MODE_NOTDEFINED:		
		resetAndDisable(alg:=algoritms.Auto_Avom_);
		resetAndDisable(alg:=algoritms.autoNu_1);
		resetAndDisable(alg:=algoritms.autoNu_2);
		resetAndDisable(alg:=algoritms.autoPns);
		resetAndDisable(alg:=algoritms.AUto_Ten_);
		resetAndDisable(alg:=algoritms.PNS_ON_MV_);
		resetAndDisable(alg:=algoritms.no);
		resetAndDisable(alg:=algoritms.ao);
		resetAndDisable(alg:=algoritms.Opres);
		resetAndDisable(alg:=algoritms.Pms);
		resetAndDisable(alg:=algoritms.dPmg);
		resetAndDisable(alg:=algoritms.ppu);
		resetAndDisable(alg:=algoritms.F1_1);
		resetAndDisable(alg:=algoritms.F1_2);
		resetAndDisable(alg:=algoritms.F2_Ch);
		resetAndDisable(alg:=algoritms.F2_R);
		resetAndDisable(alg:=algoritms.F3);
		resetAndDisable(alg:=algoritms.F4);
		resetAndDisable(alg:=algoritms.Kr6_Move);
		resetAndDisable(alg:=algoritms.AutoPNS_Start);
		resetAndDisable(alg:=algoritms.R_AutoAVom);
		resetAndDisable(alg:=algoritms.R_AutoTEN);
		resetAndDisable(alg:=algoritms.R_TestIM);
		resetAndDisable(alg:=algoritms.S_AutoAVOM);
		resetAndDisable(alg:=algoritms.S_AutoTEN);
		resetAndDisable(alg:=algoritms.S_Test_IM);
		resetAndDisable(alg:=algoritms.S_Vibr);
		resetAndDisable(alg:=algoritms.S_dPmg);
		resetAndDisable(alg:=algoritms.S_I);
		resetAndDisable(alg:=algoritms.S_K);
		resetAndDisable(alg:=algoritms.S_Pms);
		resetAndDisable(alg:=algoritms.S_V);
		resetAndDisable(alg:=algoritms.S_AP);
		resetAndDisable(alg:=algoritms.S_PP);
		resetAndDisable(alg:=algoritms.S_NO);
		resetAndDisable(alg:=algoritms.S_AO);
		resetAndDisable(alg:=algoritms.Test_IM);
		resetAndDisable(alg:=algoritms.Start_Test_P);
	resetAndDisable(alg:=algoritms.Test_P);
MODE_TESTIM:
		resetAndDisable(alg:=algoritms.Auto_Avom_);
		resetAndDisable(alg:=algoritms.autoNu_1);
		resetAndDisable(alg:=algoritms.autoNu_2);
		resetAndDisable(alg:=algoritms.autoPns);
		resetAndDisable(alg:=algoritms.AUto_Ten_);
		resetAndDisable(alg:=algoritms.PNS_ON_MV_);
		resetAndDisable(alg:=algoritms.Opres);
		resetAndDisable(alg:=algoritms.Pms);
		resetAndDisable(alg:=algoritms.dPmg);
		resetAndDisable(alg:=algoritms.no);
		resetAndDisable(alg:=algoritms.ao);
		resetAndDisable(alg:=algoritms.ppu);
		resetAndDisable(alg:=algoritms.F1_1);
		resetAndDisable(alg:=algoritms.F1_2);
		resetAndDisable(alg:=algoritms.F2_Ch);
		resetAndDisable(alg:=algoritms.F2_R);
		resetAndDisable(alg:=algoritms.F3);
		resetAndDisable(alg:=algoritms.F4);
		resetAndDisable(alg:=algoritms.Kr6_Move);
		resetAndDisable(alg:=algoritms.AutoPNS_Start);
		resetAndDisable(alg:=algoritms.R_AutoAVom);
		resetAndDisable(alg:=algoritms.R_AutoTEN);
		algoritms.R_TestIM.CanRun:=TRUE;
		resetAndDisable(alg:=algoritms.S_AutoAVOM);
		resetAndDisable(alg:=algoritms.S_AutoTEN);
		resetAndDisable(alg:=algoritms.S_Test_IM);
		resetAndDisable(alg:=algoritms.S_Vibr);
		resetAndDisable(alg:=algoritms.S_dPmg);
		resetAndDisable(alg:=algoritms.S_I);
		resetAndDisable(alg:=algoritms.S_K);
		resetAndDisable(alg:=algoritms.S_Pms);
		resetAndDisable(alg:=algoritms.S_V);
		resetAndDisable(alg:=algoritms.S_AP);
		resetAndDisable(alg:=algoritms.S_PP);
		algoritms.S_NO.CanRun:=TRUE;
		algoritms.S_AO.CanRun:=TRUE;
		resetAndDisable(alg:=algoritms.Start_Test_P);
		resetAndDisable(alg:=algoritms.Test_P);
MODE_PUSKV_R:
	resetAndDisable(alg:=algoritms.Auto_Avom_);
	resetAndDisable(alg:=algoritms.autoNu_1);
	resetAndDisable(alg:=algoritms.autoNu_2);
	resetAndDisable(alg:=algoritms.autoPns);
	resetAndDisable(alg:=algoritms.AUto_Ten_);
	resetAndDisable(alg:=algoritms.PNS_ON_MV_);
	resetAndDisable(alg:=algoritms.no);
		resetAndDisable(alg:=algoritms.ao);
	resetAndDisable(alg:=algoritms.Opres);
	resetAndDisable(alg:=algoritms.Pms);
	resetAndDisable(alg:=algoritms.dPmg);
	algoritms.ppu.CanRun:=TRUE;
	algoritms.ppu.run();
	resetAndDisable(alg:=algoritms.F1_2);
	resetAndDisable(alg:=algoritms.F2_Ch);
	resetAndDisable(alg:=algoritms.F2_R);
	resetAndDisable(alg:=algoritms.F3);
	resetAndDisable(alg:=algoritms.F4);
	resetAndDisable(alg:=algoritms.Kr6_Move);
	resetAndDisable(alg:=algoritms.AutoPNS_Start);
	resetAndDisable(alg:=algoritms.R_AutoAVom);
	resetAndDisable(alg:=algoritms.R_AutoTEN);
	resetAndDisable(alg:=algoritms.R_TestIM);
	resetAndDisable(alg:=algoritms.S_AutoAVOM);
	resetAndDisable(alg:=algoritms.S_AutoTEN);
	resetAndDisable(alg:=algoritms.S_Test_IM);
	resetAndDisable(alg:=algoritms.S_Vibr);
	resetAndDisable(alg:=algoritms.S_dPmg);
	resetAndDisable(alg:=algoritms.S_I);
	resetAndDisable(alg:=algoritms.S_K);
	resetAndDisable(alg:=algoritms.S_Pms);
	algoritms.S_V.CanRun:=FALSE;
	resetAndDisable(alg:=algoritms.S_PP);
	resetAndDisable(alg:=algoritms.S_AP);
	algoritms.S_NO.CanRun:=TRUE;
	algoritms.S_AO.CanRun:=TRUE;
	resetAndDisable(alg:=algoritms.Test_IM);
	reg_V:=TRUE;
	resetAndDisable(alg:=algoritms.Start_Test_P);
		resetAndDisable(alg:=algoritms.Test_P);
MODE_PUSKV_Ch:
	resetAndDisable(alg:=algoritms.Auto_Avom_);
	resetAndDisable(alg:=algoritms.autoNu_1);
	resetAndDisable(alg:=algoritms.autoNu_2);
	resetAndDisable(alg:=algoritms.autoPns);
	resetAndDisable(alg:=algoritms.AUto_Ten_);
	resetAndDisable(alg:=algoritms.PNS_ON_MV_);
	resetAndDisable(alg:=algoritms.no);
		resetAndDisable(alg:=algoritms.ao);
	resetAndDisable(alg:=algoritms.Opres);
	resetAndDisable(alg:=algoritms.Pms);
	resetAndDisable(alg:=algoritms.dPmg);
	algoritms.ppu.CanRun:=TRUE;
	algoritms.ppu.run();
	resetAndDisable(alg:=algoritms.F1_2);
	resetAndDisable(alg:=algoritms.F2_Ch);
	resetAndDisable(alg:=algoritms.F2_R);
	resetAndDisable(alg:=algoritms.F3);
	resetAndDisable(alg:=algoritms.F4);
	resetAndDisable(alg:=algoritms.Kr6_Move);
	resetAndDisable(alg:=algoritms.AutoPNS_Start);
	resetAndDisable(alg:=algoritms.R_AutoAVom);
	resetAndDisable(alg:=algoritms.R_AutoTEN);
	resetAndDisable(alg:=algoritms.R_TestIM);
	resetAndDisable(alg:=algoritms.S_AutoAVOM);
	resetAndDisable(alg:=algoritms.S_AutoTEN);
	resetAndDisable(alg:=algoritms.S_Test_IM);
	resetAndDisable(alg:=algoritms.S_Vibr);
	resetAndDisable(alg:=algoritms.S_dPmg);
	resetAndDisable(alg:=algoritms.S_I);
	resetAndDisable(alg:=algoritms.S_K);
	resetAndDisable(alg:=algoritms.S_Pms);
	algoritms.S_V.CanRun:=FALSE;
	resetAndDisable(alg:=algoritms.S_PP);
	resetAndDisable(alg:=algoritms.S_AP);
	algoritms.S_NO.CanRun:=TRUE;
	algoritms.S_AO.CanRun:=TRUE;
	resetAndDisable(alg:=algoritms.Test_IM);
	reg_V:=TRUE;
	resetAndDisable(alg:=algoritms.Start_Test_P);
		resetAndDisable(alg:=algoritms.Test_P);
MODE_PUSKK:
	resetAndDisable(alg:=algoritms.Auto_Avom_);
	resetAndDisable(alg:=algoritms.autoNu_1);
	resetAndDisable(alg:=algoritms.autoNu_2);
	resetAndDisable(alg:=algoritms.autoPns);
	resetAndDisable(alg:=algoritms.AUto_Ten_);
	resetAndDisable(alg:=algoritms.PNS_ON_MV_);
	resetAndDisable(alg:=algoritms.no);
		resetAndDisable(alg:=algoritms.ao);
	resetAndDisable(alg:=algoritms.Opres);
	resetAndDisable(alg:=algoritms.Pms);
	resetAndDisable(alg:=algoritms.dPmg);
	algoritms.ppu.CanRun:=TRUE;
	algoritms.ppu.run();
	resetAndDisable(alg:=algoritms.F1_2);
	resetAndDisable(alg:=algoritms.F2_Ch);
	resetAndDisable(alg:=algoritms.F2_R);
	resetAndDisable(alg:=algoritms.F3);
	resetAndDisable(alg:=algoritms.F4);
	resetAndDisable(alg:=algoritms.Kr6_Move);
	resetAndDisable(alg:=algoritms.AutoPNS_Start);
	resetAndDisable(alg:=algoritms.R_AutoAVom);
	resetAndDisable(alg:=algoritms.R_AutoTEN);
	resetAndDisable(alg:=algoritms.R_TestIM);
	resetAndDisable(alg:=algoritms.S_AutoAVOM);
	resetAndDisable(alg:=algoritms.S_AutoTEN);
	resetAndDisable(alg:=algoritms.S_Test_IM);
	resetAndDisable(alg:=algoritms.S_Vibr);
	resetAndDisable(alg:=algoritms.S_dPmg);
	resetAndDisable(alg:=algoritms.S_I);
	algoritms.S_K.CanRun:=FALSE;
	resetAndDisable(alg:=algoritms.S_Pms);
	resetAndDisable(alg:=algoritms.S_V);
	resetAndDisable(alg:=algoritms.S_PP);
	resetAndDisable(alg:=algoritms.S_AP);
	algoritms.S_NO.CanRun:=TRUE;
	algoritms.S_AO.CanRun:=TRUE;
	resetAndDisable(alg:=algoritms.Test_IM);
	resetAndDisable(alg:=algoritms.Start_Test_P);
		resetAndDisable(alg:=algoritms.Test_P);
MODE_PROVPMS:
	resetAndDisable(alg:=algoritms.Auto_Avom_);
	resetAndDisable(alg:=algoritms.autoNu_1);
	resetAndDisable(alg:=algoritms.autoNu_2);
	resetAndDisable(alg:=algoritms.autoPns);
	resetAndDisable(alg:=algoritms.AUto_Ten_);
	resetAndDisable(alg:=algoritms.PNS_ON_MV_);
	resetAndDisable(alg:=algoritms.no);
		resetAndDisable(alg:=algoritms.ao);
	resetAndDisable(alg:=algoritms.Opres);
	resetAndDisable(alg:=algoritms.Pms);
	resetAndDisable(alg:=algoritms.dPmg);
	resetAndDisable(alg:=algoritms.ppu);
	resetAndDisable(alg:=algoritms.F1_2);
	resetAndDisable(alg:=algoritms.F2_Ch);
	resetAndDisable(alg:=algoritms.F2_R);
	resetAndDisable(alg:=algoritms.F3);
	resetAndDisable(alg:=algoritms.F4);
	resetAndDisable(alg:=algoritms.Kr6_Move);
	resetAndDisable(alg:=algoritms.AutoPNS_Start);
	resetAndDisable(alg:=algoritms.R_AutoAVom);
	resetAndDisable(alg:=algoritms.R_AutoTEN);
	resetAndDisable(alg:=algoritms.R_TestIM);
	resetAndDisable(alg:=algoritms.S_AutoAVOM);
	resetAndDisable(alg:=algoritms.S_AutoTEN);
	resetAndDisable(alg:=algoritms.S_Test_IM);
	resetAndDisable(alg:=algoritms.S_Vibr);
	resetAndDisable(alg:=algoritms.S_dPmg);
	resetAndDisable(alg:=algoritms.S_I);
	resetAndDisable(alg:=algoritms.S_K);
	algoritms.S_Pms.CanRun:=FALSE;
	resetAndDisable(alg:=algoritms.S_V);
	resetAndDisable(alg:=algoritms.S_PP);
	resetAndDisable(alg:=algoritms.S_AP);
	algoritms.S_NO.CanRun:=TRUE;
	algoritms.S_AO.CanRun:=TRUE;
	resetAndDisable(alg:=algoritms.Test_IM);
	resetAndDisable(alg:=algoritms.Start_Test_P);
		resetAndDisable(alg:=algoritms.Test_P);
MODE_PROBDPMG:
	resetAndDisable(alg:=algoritms.Auto_Avom_);
	resetAndDisable(alg:=algoritms.autoNu_1);
	resetAndDisable(alg:=algoritms.autoNu_2);
	resetAndDisable(alg:=algoritms.autoPns);
	resetAndDisable(alg:=algoritms.AUto_Ten_);
	resetAndDisable(alg:=algoritms.PNS_ON_MV_);
	resetAndDisable(alg:=algoritms.no);
		resetAndDisable(alg:=algoritms.ao);
	resetAndDisable(alg:=algoritms.Opres);
	resetAndDisable(alg:=algoritms.Pms);
	resetAndDisable(alg:=algoritms.dPmg);
	resetAndDisable(alg:=algoritms.ppu);
	resetAndDisable(alg:=algoritms.F1_2);
	resetAndDisable(alg:=algoritms.F2_Ch);
	resetAndDisable(alg:=algoritms.F2_R);
	resetAndDisable(alg:=algoritms.F3);
	resetAndDisable(alg:=algoritms.F4);
	resetAndDisable(alg:=algoritms.Kr6_Move);
	resetAndDisable(alg:=algoritms.AutoPNS_Start);
	resetAndDisable(alg:=algoritms.R_AutoAVom);
	resetAndDisable(alg:=algoritms.R_AutoTEN);
	resetAndDisable(alg:=algoritms.R_TestIM);
	resetAndDisable(alg:=algoritms.S_AutoAVOM);
	resetAndDisable(alg:=algoritms.S_AutoTEN);
	resetAndDisable(alg:=algoritms.S_Test_IM);
	resetAndDisable(alg:=algoritms.S_Vibr);
	resetAndDisable(alg:=algoritms.S_Pms);
	resetAndDisable(alg:=algoritms.S_I);
	resetAndDisable(alg:=algoritms.S_K);
	algoritms.S_dPmg.CanRun:=FALSE;
	resetAndDisable(alg:=algoritms.S_V);
	resetAndDisable(alg:=algoritms.S_PP);
	resetAndDisable(alg:=algoritms.S_AP);
	algoritms.S_NO.CanRun:=TRUE;
	algoritms.S_AO.CanRun:=TRUE;
	resetAndDisable(alg:=algoritms.Test_IM);
resetAndDisable(alg:=algoritms.Start_Test_P);
		resetAndDisable(alg:=algoritms.Test_P);
MODE_I:
	resetAndDisable(alg:=algoritms.Auto_Avom_);
	resetAndDisable(alg:=algoritms.autoNu_1);
	resetAndDisable(alg:=algoritms.autoNu_2);
	resetAndDisable(alg:=algoritms.autoPns);
	resetAndDisable(alg:=algoritms.AUto_Ten_);
	resetAndDisable(alg:=algoritms.PNS_ON_MV_);
	resetAndDisable(alg:=algoritms.no);
		resetAndDisable(alg:=algoritms.ao);
	resetAndDisable(alg:=algoritms.Opres);
	resetAndDisable(alg:=algoritms.Pms);
	resetAndDisable(alg:=algoritms.dPmg);
	algoritms.ppu.CanRun:=TRUE;
	algoritms.ppu.run();
	resetAndDisable(alg:=algoritms.F1_2);
	resetAndDisable(alg:=algoritms.F2_Ch);
	resetAndDisable(alg:=algoritms.F2_R);
	resetAndDisable(alg:=algoritms.F3);
	resetAndDisable(alg:=algoritms.F4);
	resetAndDisable(alg:=algoritms.Kr6_Move);
	resetAndDisable(alg:=algoritms.AutoPNS_Start);
	resetAndDisable(alg:=algoritms.R_AutoAVom);
	resetAndDisable(alg:=algoritms.R_AutoTEN);
	resetAndDisable(alg:=algoritms.R_TestIM);
	resetAndDisable(alg:=algoritms.S_AutoAVOM);
	resetAndDisable(alg:=algoritms.S_AutoTEN);
	resetAndDisable(alg:=algoritms.S_Test_IM);
	resetAndDisable(alg:=algoritms.S_Vibr);
	resetAndDisable(alg:=algoritms.S_Pms);
	resetAndDisable(alg:=algoritms.S_dPmg);
	resetAndDisable(alg:=algoritms.S_K);
	algoritms.S_I.CanRun:=FALSE;
	resetAndDisable(alg:=algoritms.S_V);
	resetAndDisable(alg:=algoritms.S_PP);
	resetAndDisable(alg:=algoritms.S_AP);
	algoritms.S_NO.CanRun:=TRUE;
	algoritms.S_AO.CanRun:=TRUE;
	resetAndDisable(alg:=algoritms.Test_IM);
	resetAndDisable(alg:=algoritms.Start_Test_P);
		resetAndDisable(alg:=algoritms.Test_P);
MODE_O:
	resetAndDisable(alg:=algoritms.Auto_Avom_);
	resetAndDisable(alg:=algoritms.autoNu_1);
	resetAndDisable(alg:=algoritms.autoNu_2);
	resetAndDisable(alg:=algoritms.autoPns);
	resetAndDisable(alg:=algoritms.AUto_Ten_);
	resetAndDisable(alg:=algoritms.PNS_ON_MV_);
	resetAndDisable(alg:=algoritms.no);
		resetAndDisable(alg:=algoritms.ao);
	resetAndDisable(alg:=algoritms.S_I);
	resetAndDisable(alg:=algoritms.Pms);
	resetAndDisable(alg:=algoritms.dPmg);
	resetAndDisable(alg:=algoritms.ppu);
	resetAndDisable(alg:=algoritms.F1_1);
	resetAndDisable(alg:=algoritms.F1_2);
	resetAndDisable(alg:=algoritms.F2_Ch);
	resetAndDisable(alg:=algoritms.F2_R);
	resetAndDisable(alg:=algoritms.F3);
	resetAndDisable(alg:=algoritms.F4);
	resetAndDisable(alg:=algoritms.Kr6_Move);
	resetAndDisable(alg:=algoritms.AutoPNS_Start);
	resetAndDisable(alg:=algoritms.R_AutoAVom);
	resetAndDisable(alg:=algoritms.R_AutoTEN);
	resetAndDisable(alg:=algoritms.R_TestIM);
	resetAndDisable(alg:=algoritms.S_AutoAVOM);
	resetAndDisable(alg:=algoritms.S_AutoTEN);
	resetAndDisable(alg:=algoritms.S_Test_IM);
	resetAndDisable(alg:=algoritms.S_Vibr);
	resetAndDisable(alg:=algoritms.S_Pms);
	resetAndDisable(alg:=algoritms.S_dPmg);
	resetAndDisable(alg:=algoritms.S_K);
	algoritms.Opres.CanRun:=FALSE;
	resetAndDisable(alg:=algoritms.S_V);
	resetAndDisable(alg:=algoritms.S_PP);
	resetAndDisable(alg:=algoritms.S_AP);
	algoritms.S_NO.CanRun:=TRUE;
	algoritms.S_AO.CanRun:=TRUE;
	resetAndDisable(alg:=algoritms.Test_IM);
	resetAndDisable(alg:=algoritms.Start_Test_P);
		resetAndDisable(alg:=algoritms.Test_P);
		
TEST_PROTECTIONS:	
		resetAndDisable(alg:=algoritms.Auto_Avom_);
		resetAndDisable(alg:=algoritms.autoNu_1);
		resetAndDisable(alg:=algoritms.autoNu_2);
		resetAndDisable(alg:=algoritms.autoPns);
		resetAndDisable(alg:=algoritms.AUto_Ten_);
		resetAndDisable(alg:=algoritms.PNS_ON_MV_);
		algoritms.no.CanRun:=TRUE;
		algoritms.ao.CanRun:=TRUE;
		resetAndDisable(alg:=algoritms.Opres);
		resetAndDisable(alg:=algoritms.Pms);
		resetAndDisable(alg:=algoritms.dPmg);
		resetAndDisable(alg:=algoritms.ppu);
		resetAndDisable(alg:=algoritms.F1_1);
		resetAndDisable(alg:=algoritms.F1_2);
		resetAndDisable(alg:=algoritms.F2_Ch);
		resetAndDisable(alg:=algoritms.F2_R);
		resetAndDisable(alg:=algoritms.F3);
		resetAndDisable(alg:=algoritms.F4);
		resetAndDisable(alg:=algoritms.Kr6_Move);
		resetAndDisable(alg:=algoritms.AutoPNS_Start);
		resetAndDisable(alg:=algoritms.R_AutoAVom);
		resetAndDisable(alg:=algoritms.R_AutoTEN);
		resetAndDisable(alg:=algoritms.R_TestIM);
		resetAndDisable(alg:=algoritms.S_AutoAVOM);
		resetAndDisable(alg:=algoritms.S_AutoTEN);
		resetAndDisable(alg:=algoritms.S_Test_IM);
		resetAndDisable(alg:=algoritms.S_Vibr);
		resetAndDisable(alg:=algoritms.S_dPmg);
		resetAndDisable(alg:=algoritms.S_I);
		resetAndDisable(alg:=algoritms.S_K);
		resetAndDisable(alg:=algoritms.S_Pms);
		resetAndDisable(alg:=algoritms.S_V);
		resetAndDisable(alg:=algoritms.S_AP);
		resetAndDisable(alg:=algoritms.S_PP);
		algoritms.S_NO.CanRun:=TRUE;
		algoritms.S_AO.CanRun:=TRUE;
		resetAndDisable(alg:=algoritms.Test_IM);
		Reset_ALL_P ();
		resetAndDisable(alg:=algoritms.Start_Test_P);
		algoritms.Test_P.CanRun:=TRUE;
		algoritms.Test_P.EnableOpcControl();

END_CASE

END_IF
END_METHOD

METHOD PUBLIC resetAndDisable
VAR_INPUT
	alg:REFERENCE TO BaseAlgoritm;
END_VAR
IF __ISVALIDREF(alg) THEN
	IF alg.isRuning THEN
		alg.reset();
	END_IF
	alg.CanRun:=FALSE;
END_IF
END_METHOD

END_FUNCTION_BLOCK

// lowLevel_ecl/algoritms/BaseAlgoritmsManager
	{attribute 'symbol' := 'none'}
FUNCTION_BLOCK BaseAlgoritmsManager EXTENDS BaseAlgoritm
VAR_INPUT
END_VAR
VAR_OUTPUT
END_VAR
VAR

END_VAR

SUPER^();
callBase();

METHOD PROTECTED onInit
VAR_INPUT
END_VAR
SUPER^.onInit();
onStart();
END_METHOD

METHOD PROTECTED onStart
VAR_INPUT
END_VAR
END_METHOD

METHOD PROTECTED processCmd;
VAR_INPUT
	cmd:UINT;
	sender:UINT;
	parametr:UINT;
END_VAR
END_METHOD

END_FUNCTION_BLOCK

// K1/std12k5/Narabotka/NO
	{attribute 'symbol' := 'none'}
FUNCTION_BLOCK NO EXTENDS BaseIM
VAR_INPUT
END_VAR
VAR_OUTPUT
	
		{attribute 'symbol' := 'read'}
	narabotka:UDINT;
END_VAR
VAR
	flag:BOOL;
	Work_END:F_TRIG;
	
	AvomStartted:R_TRIG;
END_VAR

SUPER^();
Work_END (CLK:=(algmanager.mode=modegpa.MODE_WORK_K OR algmanager.mode=modegpa.MODE_WORK_M));
IF Work_END.Q THEN
	flag:=TRUE;
END_IF
AvomStartted(CLK:=(algmanager.mode=modegpa.MODE_NO) AND flag);
IF AvomStartted.Q THEN
	narabotka:= narabotka + 1;
	SaveToFile();
	flag:=FALSE;
END_IF

METHOD PROTECTED readPersistent
VAR_INPUT
END_VAR

narabotka:=STRING_TO_UDINT(readValue());
END_METHOD

METHOD PROTECTED writePersistent
VAR_INPUT
END_VAR

writeValue(value:= UDINT_TO_STRING(narabotka),'Наработка');
END_METHOD

END_FUNCTION_BLOCK

// K2/std12k5/Natabotka/NO
	{attribute 'symbol' := 'none'}
FUNCTION_BLOCK NO EXTENDS BaseIM
VAR_INPUT
END_VAR
VAR_OUTPUT
	
		{attribute 'symbol' := 'read'}
	narabotka:UDINT;
END_VAR
VAR
	flag:BOOL;
	Work_END:F_TRIG;
	
	AvomStartted:R_TRIG;
END_VAR

SUPER^();
Work_END (CLK:=(algmanager.mode=modegpa.MODE_WORK_K OR algmanager.mode=modegpa.MODE_WORK_M));
IF Work_END.Q THEN
	flag:=TRUE;
END_IF
AvomStartted(CLK:=(algmanager.mode=modegpa.MODE_NO) AND flag);
IF AvomStartted.Q THEN
	narabotka:= narabotka + 1;
	SaveToFile();
	flag:=FALSE;
END_IF

METHOD PROTECTED readPersistent
VAR_INPUT
END_VAR

narabotka:=STRING_TO_UDINT(readValue());
END_METHOD

METHOD PROTECTED writePersistent
VAR_INPUT
END_VAR

writeValue(value:= UDINT_TO_STRING(narabotka),'Наработка');
END_METHOD

END_FUNCTION_BLOCK

// K1/std12k5/Narabotka/AO
	{attribute 'symbol' := 'none'}
FUNCTION_BLOCK AO EXTENDS BaseIM
VAR_INPUT
END_VAR
VAR_OUTPUT
	
		{attribute 'symbol' := 'read'}
	narabotka:UDINT;
END_VAR
VAR
	Work_End:F_TRIG;
	flag:bool;
	
	AvomStartted:R_TRIG;
END_VAR

SUPER^();
Work_END (CLK:=(algmanager.mode=modegpa.MODE_WORK_K OR algmanager.mode=modegpa.MODE_WORK_M));
IF Work_END.Q THEN
	flag:=TRUE;
END_IF
AvomStartted(CLK:=(algmanager.mode=modegpa.MODE_AO) AND flag);
IF AvomStartted.Q THEN
	narabotka:= narabotka + 1;
	SaveToFile();
	flag:=false;
END_IF

METHOD PROTECTED readPersistent
VAR_INPUT
END_VAR

narabotka:=STRING_TO_UDINT(readValue());
END_METHOD

METHOD PROTECTED writePersistent
VAR_INPUT
END_VAR

writeValue(value:= UDINT_TO_STRING(narabotka),'Наработка');
END_METHOD

END_FUNCTION_BLOCK

// K2/std12k5/Natabotka/AO
	{attribute 'symbol' := 'none'}
FUNCTION_BLOCK AO EXTENDS BaseIM
VAR_INPUT
END_VAR
VAR_OUTPUT
	
		{attribute 'symbol' := 'read'}
	narabotka:UDINT;
END_VAR
VAR
	Work_End:F_TRIG;
	flag:bool;
	
	AvomStartted:R_TRIG;
END_VAR

SUPER^();
Work_END (CLK:=(algmanager.mode=modegpa.MODE_WORK_K OR algmanager.mode=modegpa.MODE_WORK_M));
IF Work_END.Q THEN
	flag:=TRUE;
END_IF
AvomStartted(CLK:=(algmanager.mode=modegpa.MODE_AO) AND flag);
IF AvomStartted.Q THEN
	narabotka:= narabotka + 1;
	SaveToFile();
	flag:=false;
END_IF

METHOD PROTECTED readPersistent
VAR_INPUT
END_VAR

narabotka:=STRING_TO_UDINT(readValue());
END_METHOD

METHOD PROTECTED writePersistent
VAR_INPUT
END_VAR

writeValue(value:= UDINT_TO_STRING(narabotka),'Наработка');
END_METHOD

END_FUNCTION_BLOCK

// K2/std12k5/Prov/Reset_ALL_P
FUNCTION Reset_ALL_P : BOOL
VAR_INPUT
END_VAR
VAR
END_VAR


		Protections.p_TOpornogoPodshipnikaEDT_1.reset ();
		Protections.p_TOpornoYpornogoPodshipnikaEDT_2.reset ();
		Protections.p_TOpornoYpornogoPodshipnikaKolesaRedEDT_3.reset ();
		Protections.p_TOpornoYpornogoPodshipnikaKolesaRedHT_4.reset ();
		Protections.p_TOpornogoPodshipnikaShesterniReduktoraT_5.reset ();
		Protections.p_TOpornogoPodshipnikaReduktoraHT_6.reset ();
		Protections.p_TOpornoYpornogoPodshipnikaNagnetateljaT_7.reset ();
		Protections.p_TOpornoYpornogoPodshipnikaSvobodnogoKoncaNT_8.reset ();
		Protections.p_TYpornogoPodshipnikaRavKolodokHT_9.reset ();
		Protections.p_TYpornogoPodshipnikaNerabKolodokHT_10.reset ();
		Protections.p_TgazaNaVyhodeH.reset ();
		
	(*Давления*)
		
		Protections.p_OsSdvigNagnetatelja_Plus.reset ();
		Protections.p_OsSdvigNagnetatelja_Minus.reset ();
		Protections.p_DGazaNaVhodeNagnetatelja_GPA_STOP.reset ();
		Protections.p_DGazaNaVyhodeNagnetatelja_GPA_STOP.reset ();
		//p_DGazaNaVhodeNagnetatelja:AiProtection (table:=protectManager.getTable())							:=(ai:=ai.DGazaNaVhodeNagnetatelja,controlLimit:=statusAi.LA,delay:=(value:=T#3S));
		Protections.p_DGazaNaVyhodeNagnetatelja.reset ();
		Protections.p_PerepadDavlenieMasloGaz.reset ();
		Protections.p_DavlenijaMasloSmNizkoe.reset ();
		Protections.p_DavlenijaMasloSmVysokoe.reset ();
	
	(*Вибрация*)
		
		Protections.p_VibroSkorostOPED_T1.reset ();
		Protections.p_VibroSkorostOYPED_T2.reset ();
		Protections.p_VibroSkorostOYPKolesaED_T3.reset ();
		Protections.p_VibroSkorostOPKolesaRH_T4.reset ();
		Protections.p_VibroSkorostOPShesterniRED_T5.reset ();
		Protections.p_VibroSkorostOPShesterniReduktoraH_T6.reset ();
	(*Дискретные сигналы *)
		
		Protections.p_PerepadDavlenieMasloGaz_Less100.reset ();
		Protections.p_RegVozbOff.reset ();
		Protections.p_Fail_Chastotniy_Pusk.reset ();
		Protections.p_OFFAvarSwitch.reset ();
		Protections.p_AOKC_SHKC.reset ();
		Protections.p_AO_PRU.reset ();
		Protections.p_AO_fromSHU.reset ();
					
(*Защиты по ИМ *)																							
		Protections.p_mvOff.reset ();
		Protections.p_kran1.reset ();
		Protections.p_kran2.reset ();

END_FUNCTION

// LowLevel_Algoritms/algoritms/AiProtection
	{attribute 'symbol' := 'none'}
FUNCTION_BLOCK AiProtection EXTENDS BaseProtection
VAR_INPUT
	ai:REFERENCE TO AISource;
	controlLimit:statusAi;
	ControlValue:REAL;
	{attribute 'symbol' := 'read'}
	delay:TimeParametr(table:=ADR(objectTable));	
END_VAR
VAR_OUTPUT
END_VAR
VAR
	flag:bool;
	timer:TON;
	timer2:ton;
END_VAR

SUPER^();
IF __ISVALIDREF(ai) THEN
	IF	((ai.interval = controlLimit) AND (ControlValue = 0)) OR ((ai.interval >= controlLimit) AND (ControlValue <> 0)) THEN
		flag:=TRUE;
	ELSE
		flag:=FALSE;
	END_IF
	IF	ControlValue <> 0 THEN
		timer2 (in:= (flag AND (ai.value >= ControlValue)), pt:=delay.Value);
		IF	timer2.Q THEN
			signaling:=TRUE;
		ELSE
			signaling:=FALSE;
		END_IF
	ELSE
		timer(IN:=flag,PT:=delay.Value);
		IF timer.Q THEN
			signaling:=TRUE;
		ELSE
			signaling:=FALSE;
		END_IF
	END_IF
END_IF

METHOD PUBLIC reset
VAR_INPUT
END_VAR
SUPER^.reset();
timer(in:=FALSE);
signaling:=FALSE;
DisableAiLimits( ai,getLimitFlags(controlLimit));
END_METHOD

METHOD PUBLIC run
VAR_INPUT
END_VAR
SUPER^.run();
EnableAiLimits( ai,getLimitFlags(controlLimit));
END_METHOD

END_FUNCTION_BLOCK

// LowLevel_Algoritms/Common/DisableAiLimits
FUNCTION DisableAiLimits : Bool
VAR_INPUT
	ai:REFERENCE TO AISource;
	flags:BYTE;
END_VAR
VAR
END_VAR

IF __ISVALIDREF(ai) THEN
	ai.disabledAlarms:=ai.disabledAlarms OR flags;
END_IF

END_FUNCTION

// LowLevel_Algoritms/Common/getLimitFlags
FUNCTION getLimitFlags : BYTE
VAR_INPUT
	AiLimit:statusAi;
END_VAR
VAR
END_VAR

CASE AiLimit OF
	statusAi.LW, statusAi.LA:
		getLimitFlags:=AnalogAlarms.LW OR AnalogAlarms.LA;
	statusAi.HW,statusAi.HA:
		getLimitFlags:=AnalogAlarms.HW OR AnalogAlarms.HA;
ELSE
	getLimitFlags:=0;
END_CASE

END_FUNCTION

// LowLevel_Algoritms/Common/EnableAiLimits
FUNCTION EnableAiLimits : Bool
VAR_INPUT
	ai:REFERENCE TO AISource;
	flags:BYTE;
END_VAR
VAR
END_VAR

IF __ISVALIDREF(ai) THEN
	ai.disabledAlarms:=ai.disabledAlarms AND (flags XOR 16#FF);
END_IF

END_FUNCTION

// K1/std12k5/Prov/Reset_ALL_P
FUNCTION Reset_ALL_P : BOOL
VAR_INPUT
END_VAR
VAR
END_VAR


		Protections.p_TOpornogoPodshipnikaEDT_1.reset ();
		Protections.p_TOpornoYpornogoPodshipnikaEDT_2.reset ();
		Protections.p_TOpornoYpornogoPodshipnikaKolesaRedEDT_3.reset ();
		Protections.p_TOpornoYpornogoPodshipnikaKolesaRedHT_4.reset ();
		Protections.p_TOpornogoPodshipnikaShesterniReduktoraT_5.reset ();
		Protections.p_TOpornogoPodshipnikaReduktoraHT_6.reset ();
		Protections.p_TOpornoYpornogoPodshipnikaNagnetateljaT_7.reset ();
		Protections.p_TOpornoYpornogoPodshipnikaSvobodnogoKoncaNT_8.reset ();
		Protections.p_TYpornogoPodshipnikaRavKolodokHT_9.reset ();
		Protections.p_TYpornogoPodshipnikaNerabKolodokHT_10.reset ();
		Protections.p_TgazaNaVyhodeH.reset ();
		
	(*Давления*)
		
		Protections.p_OsSdvigNagnetatelja_Plus.reset ();
		Protections.p_OsSdvigNagnetatelja_Minus.reset ();
		Protections.p_DGazaNaVhodeNagnetatelja_GPA_STOP.reset ();
		Protections.p_DGazaNaVyhodeNagnetatelja_GPA_STOP.reset ();
		//p_DGazaNaVhodeNagnetatelja:AiProtection (table:=protectManager.getTable())							:=(ai:=ai.DGazaNaVhodeNagnetatelja,controlLimit:=statusAi.LA,delay:=(value:=T#3S));
		Protections.p_DGazaNaVyhodeNagnetatelja.reset ();
		Protections.p_PerepadDavlenieMasloGaz.reset ();
		Protections.p_DavlenijaMasloSmNizkoe.reset ();
		Protections.p_DavlenijaMasloSmVysokoe.reset ();
	
	(*Вибрация*)
		
		Protections.p_VibroSkorostOPED_T1.reset ();
		Protections.p_VibroSkorostOYPED_T2.reset ();
		Protections.p_VibroSkorostOYPKolesaED_T3.reset ();
		Protections.p_VibroSkorostOPKolesaRH_T4.reset ();
		Protections.p_VibroSkorostOPShesterniRED_T5.reset ();
		Protections.p_VibroSkorostOPShesterniReduktoraH_T6.reset ();
	(*Дискретные сигналы *)
		
		Protections.p_PerepadDavlenieMasloGaz_Less100.reset ();
		Protections.p_RegVozbOff.reset ();
		Protections.p_Fail_Chastotniy_Pusk.reset ();
		Protections.p_OFFAvarSwitch.reset ();
		Protections.p_AOKC_SHKC.reset ();
		Protections.p_AO_PRU.reset ();
		Protections.p_AO_fromSHU.reset ();
					
(*Защиты по ИМ *)																							
		Protections.p_mvOff.reset ();
		Protections.p_kran1.reset ();
		Protections.p_kran2.reset ();

END_FUNCTION

// K1/std12k5/Prov/Test_Protections
	{attribute 'symbol' := 'none'}
FUNCTION_BLOCK  Test_Protections EXTENDS BaseAlgoritm
VAR_INPUT
	{attribute 'symbol' := 'read'}
	Protect_On_1:DiscretParametr(table:=ADR(objectTable));//{name:маска ввключения защит}
	{attribute 'symbol' := 'read'}
	Protect_On_2:DiscretParametr(table:=ADR(objectTable));//{name:маска ввключения защит}
	{attribute 'symbol' := 'read'}
	Protect_On_3:DiscretParametr(table:=ADR(objectTable));//{name:маска ввключения защит}
	{attribute 'symbol' := 'read'}
	Protect_On_4:DiscretParametr(table:=ADR(objectTable));//{name:маска ввключения защит}
	{attribute 'symbol' := 'read'}
	AO_start:DiscretParametr(table:=ADR(objectTable));//{name:маска ввключения защит}
END_VAR
VAR_OUTPUT
	
END_VAR
VAR

	
	
END_VAR

SUPER^();
Run_Protection(Protections.p_TOpornogoPodshipnikaEDT_1						, 1		,Protect_On_1.value);
Run_Protection(Protections.p_TOpornoYpornogoPodshipnikaEDT_2				, 2		,Protect_On_1.value);
Run_Protection(Protections.p_TOpornoYpornogoPodshipnikaKolesaRedEDT_3  		, 4		,Protect_On_1.value);
Run_Protection(Protections.p_TOpornoYpornogoPodshipnikaKolesaRedHT_4   		, 8		,Protect_On_1.value);
Run_Protection(Protections.p_TOpornogoPodshipnikaShesterniReduktoraT_5	 	, 16	,Protect_On_1.value);
Run_Protection(Protections.p_TOpornogoPodshipnikaReduktoraHT_6	         	, 32	,Protect_On_1.value);
Run_Protection(Protections.p_TOpornoYpornogoPodshipnikaNagnetateljaT_7	 	, 64	,Protect_On_1.value);
Run_Protection(Protections.p_TOpornoYpornogoPodshipnikaSvobodnogoKoncaNT_8	, 128	,Protect_On_1.value);
Run_Protection(Protections.p_TYpornogoPodshipnikaRavKolodokHT_9				, 256	,Protect_On_1.value);
Run_Protection(Protections.p_TYpornogoPodshipnikaNerabKolodokHT_10			, 512	,Protect_On_1.value);
Run_Protection(Protections.p_TgazaNaVyhodeH									, 1		,Protect_On_2.value);
Run_Protection(Protections.p_OsSdvigNagnetatelja_Plus						, 2		,Protect_On_2.value);
Run_Protection(Protections.p_OsSdvigNagnetatelja_Minus						, 4		,Protect_On_2.value);
Run_Protection(Protections.p_DGazaNaVhodeNagnetatelja_GPA_STOP				, 8		,Protect_On_2.value);
Run_Protection(Protections.p_DGazaNaVyhodeNagnetatelja_GPA_STOP				, 16	,Protect_On_2.value);
Run_Protection(Protections.p_DGazaNaVyhodeNagnetatelja						, 32	,Protect_On_2.value);
Run_Protection(Protections.p_PerepadDavlenieMasloGaz						, 64	,Protect_On_2.value);
Run_Protection(Protections.p_DavlenijaMasloSmNizkoe							, 128	,Protect_On_2.value);
Run_Protection(Protections.p_DavlenijaMasloSmVysokoe						, 256	,Protect_On_2.value);
Run_Protection(Protections.p_VibroSkorostOPED_T1							, 512	,Protect_On_2.value);
Run_Protection(Protections.p_VibroSkorostOYPED_T2							, 1		,Protect_On_3.value);
Run_Protection(Protections.p_VibroSkorostOYPKolesaED_T3						, 2		,Protect_On_3.value);
Run_Protection(Protections.p_VibroSkorostOPKolesaRH_T4						, 4		,Protect_On_3.value);
Run_Protection(Protections.p_VibroSkorostOPShesterniRED_T5					, 8		,Protect_On_3.value);
Run_Protection(Protections.p_VibroSkorostOPShesterniReduktoraH_T6			, 16	,Protect_On_3.value);
Run_Protection(Protections.p_PerepadDavlenieMasloGaz_Less100				, 32	,Protect_On_3.value);
Run_Protection(Protections.p_RegVozbOff										, 64	,Protect_On_3.value);
Run_Protection(Protections.p_Fail_Chastotniy_Pusk							, 128	,Protect_On_3.value);
Run_Protection(Protections.p_OFFAvarSwitch									, 256	,Protect_On_3.value);
Run_Protection(Protections.p_AOKC_SHKC										, 512	,Protect_On_3.value);																				
Run_Protection(Protections.p_AO_PRU											, 1		,Protect_On_4.value);
Run_Protection(Protections.p_AO_fromSHU										, 2		,Protect_On_4.value);
Run_Protection(Protections.p_mvOff											, 4		,Protect_On_4.value);
Run_Protection(Protections.p_kran1											, 8		,Protect_On_4.value);
Run_Protection(Protections.p_kran2											, 16	,Protect_On_4.value);


		
		
		
		
		
		
		
		
		
		
		
	
	
	(*Вибрация*)
		
		
		
		
		
		
		
	(*Дискретные сигналы *)
		
		
		
		
		
		
		
		
					
(*Защиты по ИМ *)

METHOD PUBLIC reset
VAR_INPUT
END_VAR
SUPER^.reset();
Reset_All_P ();
AO_start.setValue (0);
Protect_On_1.setValue (0);
Protect_On_2.setValue (0);
Protect_On_3.setValue (0);
Protect_On_4.setValue (0);
END_METHOD

METHOD PUBLIC run
VAR_INPUT
END_VAR
SUPER^.run();
algManager.setMode	(ModeGpa.TEST_PROTECTIONS);
END_METHOD

METHOD PRIVATE Run_Protection
VAR_INPUT
	protection: REFERENCE TO  BaseProtection;
	num:UINT;
	num_bits:UINT;
END_VAR
VAR
	run_protect:R_trig;
	reset_protect:R_trig;
END_VAR

IF	__ISVALIDREF(protection) THEN
	run_protect (clk:=(((num_bits AND num)<> 0) AND NOT protection.isRuning));
	reset_protect (clk:=((num_bits AND num) = 0) AND protection.isRuning);
	IF	run_protect.Q THEN
		protection.run();
	END_IF
	IF	reset_protect.Q THEN
		protection.reset();
	END_IF
END_IF
END_METHOD

END_FUNCTION_BLOCK

// K2/std12k5/Prov/Test_Protections
	{attribute 'symbol' := 'none'}
FUNCTION_BLOCK  Test_Protections EXTENDS BaseAlgoritm
VAR_INPUT
	{attribute 'symbol' := 'read'}
	Protect_On_1:DiscretParametr(table:=ADR(objectTable));//{name:маска ввключения защит}
	{attribute 'symbol' := 'read'}
	Protect_On_2:DiscretParametr(table:=ADR(objectTable));//{name:маска ввключения защит}
	{attribute 'symbol' := 'read'}
	Protect_On_3:DiscretParametr(table:=ADR(objectTable));//{name:маска ввключения защит}
	{attribute 'symbol' := 'read'}
	Protect_On_4:DiscretParametr(table:=ADR(objectTable));//{name:маска ввключения защит}
	{attribute 'symbol' := 'read'}
	AO_start:DiscretParametr(table:=ADR(objectTable));//{name:маска ввключения защит}
END_VAR
VAR_OUTPUT
	
END_VAR
VAR

	
	
END_VAR

SUPER^();
Run_Protection(Protections.p_TOpornogoPodshipnikaEDT_1						, 1		,Protect_On_1.value);
Run_Protection(Protections.p_TOpornoYpornogoPodshipnikaEDT_2				, 2		,Protect_On_1.value);
Run_Protection(Protections.p_TOpornoYpornogoPodshipnikaKolesaRedEDT_3  		, 4		,Protect_On_1.value);
Run_Protection(Protections.p_TOpornoYpornogoPodshipnikaKolesaRedHT_4   		, 8		,Protect_On_1.value);
Run_Protection(Protections.p_TOpornogoPodshipnikaShesterniReduktoraT_5	 	, 16	,Protect_On_1.value);
Run_Protection(Protections.p_TOpornogoPodshipnikaReduktoraHT_6	         	, 32	,Protect_On_1.value);
Run_Protection(Protections.p_TOpornoYpornogoPodshipnikaNagnetateljaT_7	 	, 64	,Protect_On_1.value);
Run_Protection(Protections.p_TOpornoYpornogoPodshipnikaSvobodnogoKoncaNT_8	, 128	,Protect_On_1.value);
Run_Protection(Protections.p_TYpornogoPodshipnikaRavKolodokHT_9				, 256	,Protect_On_1.value);
Run_Protection(Protections.p_TYpornogoPodshipnikaNerabKolodokHT_10			, 512	,Protect_On_1.value);
Run_Protection(Protections.p_TgazaNaVyhodeH									, 1		,Protect_On_2.value);
Run_Protection(Protections.p_OsSdvigNagnetatelja_Plus						, 2		,Protect_On_2.value);
Run_Protection(Protections.p_OsSdvigNagnetatelja_Minus						, 4		,Protect_On_2.value);
Run_Protection(Protections.p_DGazaNaVhodeNagnetatelja_GPA_STOP				, 8		,Protect_On_2.value);
Run_Protection(Protections.p_DGazaNaVyhodeNagnetatelja_GPA_STOP				, 16	,Protect_On_2.value);
Run_Protection(Protections.p_DGazaNaVyhodeNagnetatelja						, 32	,Protect_On_2.value);
Run_Protection(Protections.p_PerepadDavlenieMasloGaz						, 64	,Protect_On_2.value);
Run_Protection(Protections.p_DavlenijaMasloSmNizkoe							, 128	,Protect_On_2.value);
Run_Protection(Protections.p_DavlenijaMasloSmVysokoe						, 256	,Protect_On_2.value);
Run_Protection(Protections.p_VibroSkorostOPED_T1							, 512	,Protect_On_2.value);
Run_Protection(Protections.p_VibroSkorostOYPED_T2							, 1		,Protect_On_3.value);
Run_Protection(Protections.p_VibroSkorostOYPKolesaED_T3						, 2		,Protect_On_3.value);
Run_Protection(Protections.p_VibroSkorostOPKolesaRH_T4						, 4		,Protect_On_3.value);
Run_Protection(Protections.p_VibroSkorostOPShesterniRED_T5					, 8		,Protect_On_3.value);
Run_Protection(Protections.p_VibroSkorostOPShesterniReduktoraH_T6			, 16	,Protect_On_3.value);
Run_Protection(Protections.p_PerepadDavlenieMasloGaz_Less100				, 32	,Protect_On_3.value);
Run_Protection(Protections.p_RegVozbOff										, 64	,Protect_On_3.value);
Run_Protection(Protections.p_Fail_Chastotniy_Pusk							, 128	,Protect_On_3.value);
Run_Protection(Protections.p_OFFAvarSwitch									, 256	,Protect_On_3.value);
Run_Protection(Protections.p_AOKC_SHKC										, 512	,Protect_On_3.value);																				
Run_Protection(Protections.p_AO_PRU											, 1		,Protect_On_4.value);
Run_Protection(Protections.p_AO_fromSHU										, 2		,Protect_On_4.value);
Run_Protection(Protections.p_mvOff											, 4		,Protect_On_4.value);
Run_Protection(Protections.p_kran1											, 8		,Protect_On_4.value);
Run_Protection(Protections.p_kran2											, 16	,Protect_On_4.value);


		
		
		
		
		
		
		
		
		
		
		
	
	
	(*Вибрация*)
		
		
		
		
		
		
		
	(*Дискретные сигналы *)
		
		
		
		
		
		
		
		
					
(*Защиты по ИМ *)

METHOD PUBLIC reset
VAR_INPUT
END_VAR
SUPER^.reset();
Reset_All_P ();
AO_start.setValue (0);
Protect_On_1.setValue (0);
Protect_On_2.setValue (0);
Protect_On_3.setValue (0);
Protect_On_4.setValue (0);
END_METHOD

METHOD PUBLIC run
VAR_INPUT
END_VAR
SUPER^.run();
algManager.setMode	(ModeGpa.TEST_PROTECTIONS);
END_METHOD

METHOD PRIVATE Run_Protection
VAR_INPUT
	protection: REFERENCE TO  BaseProtection;
	num:UINT;
	num_bits:UINT;
END_VAR
VAR
	run_protect:R_trig;
	reset_protect:R_trig;
END_VAR

IF	__ISVALIDREF(protection) THEN
	run_protect (clk:=(((num_bits AND num)<> 0) AND NOT protection.isRuning));
	reset_protect (clk:=((num_bits AND num) = 0) AND protection.isRuning);
	IF	run_protect.Q THEN
		protection.run();
	END_IF
	IF	reset_protect.Q THEN
		protection.reset();
	END_IF
END_IF
END_METHOD

END_FUNCTION_BLOCK

// lowLevel_ecl/Common/parameters/DiscretParametr
	{attribute 'symbol' := 'none'}
FUNCTION_BLOCK DiscretParametr EXTENDS BaseIm
VAR_INPUT
	
END_VAR
VAR_OUTPUT
	Value:UINT;
END_VAR
VAR
	
END_VAR
VAR CONSTANT
	cmd_ChangeValue:WORD:=1;
END_VAR


SUPER^();

METHOD PROTECTED processCmd;
VAR_INPUT
	cmd:UINT;
	sender:UINT;
	parametr:UINT;
END_VAR
CASE cmd OF
	cmd_ChangeValue:setValue(newValue:=parametr);
END_CASE
END_METHOD

METHOD PROTECTED readPersistent
VAR_INPUT
END_VAR
value:=STRING_TO_UINT(readValue());
END_METHOD

METHOD PUBLIC setValue
VAR_INPUT
	newValue:uint;
END_VAR
setCmd(cmd_ChangeValue);
Value:=newValue;
SaveToFile();

resetCommand();
END_METHOD

METHOD PUBLIC writeImStatus
VAR_INPUT
END_VAR
SUPER^.writeImStatus();
statusSet.setBits(5,14,value);
END_METHOD

METHOD PROTECTED writePersistent
VAR_INPUT
END_VAR
writeValue(value:=UINT_TO_STRING(value),comment:='value');
END_METHOD

END_FUNCTION_BLOCK

// LowLevel_Algoritms/algoritms/Krans_Protections
{attribute 'symbol' := 'none'}
FUNCTION_BLOCK PUBLIC Krans_Protections EXTENDS BaseProtection
VAR_INPUT
	Krans:	REFERENCE TO Kran;
	delay:TimeParametr(table:=ADR(objectTable));
	dP_Konf:REFERENCE TO DiscretParametr;//{name:режим работы защиты}
END_VAR
VAR_OUTPUT
END_VAR
VAR
	dP_Konf_izm:REAL;
	timer:TON;
END_VAR

SUPER^();
IF __ISVALIDREF(Krans) THEN
	IF 	(dP_Konf.Value = 0) THEN
		dP_Konf_izm:=0;	
		timer (in:=(krans.onStatus <> statusDualInput.status_on AND ((krans.onStatus = statusDualInput.status_off) OR (krans.onStatus = statusDualInput.STATUS_TRANSITIONAL))), PT:=delay.Value);
		IF	timer.Q THEN
			signaling:=TRUE;
		ELSE
			signaling:=FALSE;
		END_IF
	ELSE
		timer(in:=FALSE);
		IF	(krans.onStatus <> statusDualInput.status_on) AND ((krans.onStatus = statusDualInput.status_off) OR (krans.onStatus = statusDualInput.STATUS_TRANSITIONAL)) AND (dP_Konf_izm=0) AND (ai.PerepadDavlenieNaKonfuzore.interval >= normal) THEN
			dP_Konf_izm:=ai.PerepadDavlenieNaKonfuzore.value;
		ELSIF 	(krans.onStatus = statusDualInput.status_on) OR (ai.PerepadDavlenieNaKonfuzore.interval < normal) THEN
				dP_Konf_izm:=0;	
		END_IF
		IF	((dP_Konf_izm - ai.PerepadDavlenieNaKonfuzore.value) >= 10) AND (ai.PerepadDavlenieNaKonfuzore.interval >= normal) THEN
			signaling:=TRUE;
		ELSE
			signaling:=FALSE;
		END_IF
	END_IF
	
END_IF
(*IF	remont THEN
	timer(in:=FALSE);
	signaling:=FALSE;
	dP_Konf_izm:=0;
END_IF*)

METHOD PUBLIC reset
VAR_INPUT
END_VAR
SUPER^.reset();
timer(in:=FALSE);
signaling:=FALSE;
dP_Konf_izm:=0;
END_METHOD

END_FUNCTION_BLOCK

// lowLevel_ecl/im/Kran/Kran
	{attribute 'symbol' := 'none'}
FUNCTION_BLOCK Kran EXTENDS DualStateKran
VAR_INPUT
	inLocal: REFERENCE TO ReliableBit;	
	inDistance: REFERENCE TO ReliableBit;
	inAuto:REFERENCE TO ReliableBit;
	inManual: REFERENCE TO ReliableBit;
	
	inErrorPowerOff: REFERENCE TO ReliableBit;
	inErrorBlock: REFERENCE TO ReliableBit;	
	inSo:REFERENCE TO ReliableBit;
	inSz:REFERENCE TO ReliableBit;
	
	inDp:REFERENCE TO ReliableBit;
END_VAR
VAR_OUTPUT
	Local: BOOL;	
	Distance: BOOL;
	Auto:BOOL;
	Manual:BOOL;
	
	ErrorPowerOff: BOOL;
	ErrorBlock: BOOL;	
	So:BOOL;
	Sz:BOOL;
	
	Dp:BOOL;
END_VAR
VAR
	outputsSets:TOF:=(PT:=T#2S);
END_VAR

SUPER^();

Local:=checkArg(inLocal);
Distance:=checkArg(inDistance);
Auto:=checkArg(inAuto);
Manual:=checkArg(inManual);

ErrorPowerOff:=checkArg(inErrorPowerOff);
ErrorBlock:=checkArg(inErrorBlock);

outputsSets(in:=validAndTrue(input:=CmdOn) OR validAndTrue(input:=CmdOff));
So:=checkArg(inSo) AND NOT (outputsSets.Q);
Sz:=checkArg(inSz) AND NOT (outputsSets.Q);

Dp:=checkArg(inDp);

METHOD PROTECTED getSdvig : BOOL
VAR_INPUT
END_VAR
getSdvig:=FALSE;
IF (NOT Local) THEN
	getSdvig:=super^.getSdvig();
END_IF
END_METHOD

METHOD PUBLIC writeImStatus
VAR_INPUT
END_VAR
SUPER^.writeImStatus();
statusSet.setBit(5,Local);
statusSet.setBit(6,Distance);
statusSet.setBit(7,Auto);
statusSet.setBit(8,Manual);

statusSet.setBit(10,ErrorPowerOff);
statusSet.setBit(11,ErrorBlock);
statusSet.setBit(12,So);
statusSet.setBit(13,Sz);

statusSet.setBit(14,Dp);
END_METHOD

END_FUNCTION_BLOCK

// lowLevel_ecl/Common/functions/validAndTrue
FUNCTION validAndTrue : bool
VAR_INPUT
	input: REFERENCE TO BOOL;
END_VAR
VAR
END_VAR

IF __ISVALIDREF(input) THEN
	validAndTrue:=input;
ELSE
	validAndTrue:=FALSE;
END_IF

END_FUNCTION

// lowLevel_ecl/im/BaseIms/DualStateKran
	{attribute 'symbol' := 'none'}
FUNCTION_BLOCK DualStateKran EXTENDS DualStateIm
VAR_INPUT	
	cmdReset:REFERENCE TO BOOL;
	continueHoldCommand:TIME:=T#0S;	
END_VAR
VAR_OUTPUT

END_VAR
VAR
	_commandTimer:TON:=(PT:=T#90S);
	_resetTimer:TON:=(PT:=T#5S);
	continueHoldCommandTimer:TON;
END_VAR
VAR CONSTANT
	cmd_open:WORD:=1;
	cmd_close:WORD:=2;
	cmd_reset:WORD:=3;
END_VAR

SUPER^();

METHOD PUBLIC close
VAR_INPUT
END_VAR
off();
END_METHOD

METHOD PUBLIC off
VAR_INPUT
END_VAR
setCmd(nCmd:=cmd_close);
_commandTimer(IN:=FALSE);
_commandTimer.IN:=TRUE;
SUPER^.off();
END_METHOD

METHOD PUBLIC reset
VAR_INPUT
END_VAR
setCmd(nCmd:=cmd_reset);
_commandTimer(IN:=FALSE);
resetOuts();
IF __ISVALIDREF(cmdReset) THEN
	cmdReset:=TRUE;
	_resetTimer.IN:=TRUE;
ELSE
	resetCommand();
END_IF
END_METHOD

METHOD PUBLIC on
VAR_INPUT
END_VAR
setCmd(nCmd:=cmd_open);
_commandTimer(IN:=FALSE);
_commandTimer.IN:=TRUE;
SUPER^.on();
END_METHOD

METHOD PUBLIC open
VAR_INPUT
END_VAR
on();
END_METHOD

METHOD PRIVATE doOpenCloseCmd
VAR_INPUT
	complite:BOOL;
END_VAR
_commandTimer();

IF complite THEN
	continueHoldCommandTimer(IN:=TRUE,PT:=continueHoldCommand);
	IF continueHoldCommandTimer.Q THEN
		resetCommand();
	END_IF
ELSE
	continueHoldCommandTimer(IN:=FALSE);
	IF _commandTimer.Q THEN
		errorCommand();
	END_IF	
END_IF
END_METHOD

//Метод вызывается каждый такт пересчета пока идет выполенение команды.
METHOD PROTECTED onCommandActive
VAR_INPUT
	command:WORD;
END_VAR
CASE command OF
	cmd_open:
		doOpenCloseCmd(onStatus=statusDualInput.STATUS_ON);
	cmd_close:
		doOpenCloseCmd(onStatus=statusDualInput.STATUS_OFF);
	cmd_reset:
		IF __ISVALIDREF(cmdReset) THEN
			_resetTimer();
			IF _resetTimer.Q THEN
				cmdReset:=FALSE;
				resetCommand();
			END_IF
		END_IF
ELSE
	SUPER^.onCommandActive(command);
	RETURN;
END_CASE
END_METHOD

METHOD PROTECTED processCmd;
VAR_INPUT
	cmd:UINT;
	sender:UINT;
	parametr:UINT;
END_VAR
SUPER^.processCmd(cmd,sender,parametr);
CASE cmd OF
	cmd_open:open();
	cmd_close:close();
	cmd_reset:reset();
END_CASE
END_METHOD

METHOD PROTECTED resetCommand
VAR_INPUT
END_VAR
SUPER^.resetCommand();
_commandTimer(IN:=FALSE);
_resetTimer(In:=FALSE);
END_METHOD

END_FUNCTION_BLOCK

// lowLevel_ecl/im/BaseIms/DualStateIm
	{attribute 'symbol' := 'none'}
FUNCTION_BLOCK DualStateIm EXTENDS BaseIm
VAR_INPUT
	statOn:REFERENCE TO ReliableBit;
	statOff:REFERENCE TO ReliableBit;
	
	inAccident:REFERENCE TO ReliableBit;
	inNs:REFERENCE TO ReliableBit;
	
	CmdOn: REFERENCE TO BOOL;
	CmdOff:REFERENCE TO BOOL;
END_VAR
VAR_OUTPUT
	onStatus:statusDualInput;
	sdvig:BOOL;
	Accident:BOOL;
	Ns:BOOL;
END_VAR
VAR
	_lastCmd:INT;
	_lastStatus:statusDualInput;
	_sdvigReset:TON:=(PT:=T#15S);	
END_VAR
VAR CONSTANT
	baseCmdOn:INT:=1;
	baseCmdOff:INT:=2;
END_VAR

onStatus:=getStatus();

IF getSdvig() THEN
	sdvig:= TRUE;
END_IF
_lastStatus:=onStatus;

SUPER^();

_sdvigReset(IN:=sdvig);
IF _sdvigReset.Q THEN
	sdvig:=FALSE;
END_IF

Accident:=checkArg(inAccident);
Ns:=checkArg(inNs);

METHOD PUBLIC off
VAR_INPUT
END_VAR
IF __ISVALIDREF(CmdOff) THEN
	CmdOff:=TRUE;
	IF __ISVALIDREF(CmdOn) THEN
		CmdOn:=FALSE;		
	END_IF
ELSIF __ISVALIDREF(CmdOn) THEN
	CmdOn:=FALSE;
END_IF
_lastCmd:=baseCmdOff;
END_METHOD

METHOD PRIVATE calcStatus: statusDualInput
VAR_INPUT
	statOn:BOOL;
	statOff:BOOL;
	reliability:BOOL;
END_VAR
VAR
	on:BOOL;
	off:BOOL;
END_VAR
IF reliability THEN
	on:=statOn ;
	off:=statOff;
	IF  On AND NOT Off THEN
		calcStatus:=statusDualInput.STATUS_ON;
	ELSIF Off AND NOT On THEN
		calcStatus:=statusDualInput.Status_OFF;
	ELSIF NOT On AND NOT Off THEN
		calcStatus:=statusDualInput.STATUS_TRANSITIONAL;
	ELSE
		calcStatus:=statusDualInput.STATUS_ERROR;
	END_IF
ELSE
	calcStatus:=statusDualInput.STATUS_NOTDEFINED;
END_IF
END_METHOD

METHOD PROTECTED getSdvig : BOOL
VAR_INPUT
END_VAR
getSdvig:=FALSE;
IF (__ISVALIDREF(CmdOn)) OR ( __ISVALIDREF(CmdOff)) THEN
	IF _cmd=0 THEN
		IF (_lastStatus<>onStatus AND 
		(onStatus<>statusDualInput.STATUS_NOTDEFINED AND onStatus<>statusDualInput.STATUS_ERROR) AND
		(_lastStatus<>statusDualInput.STATUS_NOTDEFINED AND _lastStatus<>statusDualInput.STATUS_ERROR)) THEN
			getSdvig:=TRUE;
		END_IF
	END_IF
END_IF
END_METHOD

METHOD PROTECTED getStatus : statusDualInput
VAR_INPUT
END_VAR
IF __ISVALIDREF(statOn) AND __ISVALIDREF(statOff) THEN
	getStatus:=calcStatus(statOn.value,statOff.value,statOn.reliability AND statOff.reliability);
ELSIF __ISVALIDREF(statOn) THEN
	getStatus:=calcStatus(statOn.value,NOT statOn.value,statOn.reliability);
ELSIF __ISVALIDREF(statOff) THEN
	getStatus:=calcStatus(NOT statOff.value,statOff.value,statOff.reliability);
ELSE
	getStatus:=noStatusLinks();
END_IF
END_METHOD

METHOD PROTECTED onInit
VAR_INPUT
END_VAR
SUPER^.onInit();
IF (__ISVALIDREF(CmdOn) XOR __ISVALIDREF(CmdOff)) THEN
	IF 	__ISVALIDREF(CmdOn) THEN
		_lastCmd:= baseCmdOff;
	ELSE
		_lastCmd:= baseCmdOn;
	END_IF
END_IF
END_METHOD

METHOD PROTECTED resetCommand
VAR_INPUT
END_VAR
SUPER^.resetCommand();
resetOuts();
END_METHOD

METHOD PROTECTED noStatusLinks: statusDualInput
VAR_INPUT
END_VAR
CASE _lastCmd OF	
	baseCmdOn:	noStatusLinks:=statusDualInput.STATUS_ON;
	baseCmdOff: noStatusLinks:=statusDualInput.STATUS_OFF;
ELSE
	noStatusLinks:=statusDualInput.STATUS_NOTDEFINED;
END_CASE
END_METHOD

METHOD PUBLIC resetOuts
VAR_INPUT
END_VAR
IF __ISVALIDREF(CmdOn) AND __ISVALIDREF(CmdOff) THEN
	CmdOn:=FALSE;
	CmdOff:=FALSE;
END_IF;
END_METHOD

METHOD PUBLIC on
VAR_INPUT
END_VAR
IF __ISVALIDREF(CmdOn) THEN
	CmdOn:=TRUE;
	IF __ISVALIDREF(CmdOff) THEN
		CmdOff:=FALSE;		
	END_IF
ELSIF __ISVALIDREF(CmdOff) THEN
	CmdOff:=FALSE;
END_IF
_lastCmd:=baseCmdOn;
END_METHOD

METHOD PUBLIC writeImStatus
VAR_INPUT
END_VAR
SUPER^.writeImStatus();
statusSet.setBits(0,2,onStatus);
statusSet.setBit(3,Accident);
statusSet.setBit(4,Ns);
statusSet.setBit(22,sdvig);
END_METHOD

END_FUNCTION_BLOCK

// LowLevel_Algoritms/algoritms/DiProtection_fb
	{attribute 'symbol' := 'none'}
FUNCTION_BLOCK DiProtection_fb EXTENDS BaseProtection
VAR_INPUT
	FB:DWORD;
	{attribute 'symbol' := 'read'}
	delay:TimeParametr(table:=ADR(objectTable));	
END_VAR
VAR_OUTPUT
END_VAR
VAR
	timer:TON;
END_VAR

SUPER^();
timer(IN:=FB=1,PT:=delay.Value);
	IF timer.Q THEN
		signaling:=TRUE;
	ELSE
		signaling:=FALSE;
	END_IF

METHOD PUBLIC reset
VAR_INPUT
END_VAR
SUPER^.reset();
timer(in:=FALSE);
signaling:=FALSE;
END_METHOD

END_FUNCTION_BLOCK

// LowLevel_Algoritms/algoritms/DiProtection
	{attribute 'symbol' := 'none'}
FUNCTION_BLOCK DiProtection EXTENDS BaseProtection
VAR_INPUT
	di:REFERENCE TO singleSignal;
	when:BOOL:=TRUE;
	{attribute 'symbol' := 'read'}
	delay:TimeParametr(table:=ADR(objectTable));	
END_VAR
VAR_OUTPUT
END_VAR
VAR
	timer:TON;
END_VAR

SUPER^();
IF __ISVALIDREF(di) THEN
	timer(IN:=di.q=when,PT:=delay.Value);
	
	IF timer.Q THEN
		signaling:=TRUE;
	ELSE
		signaling:=FALSE;
	END_IF
END_IF

METHOD PUBLIC reset
VAR_INPUT
END_VAR
SUPER^.reset();
timer(in:=FALSE);
signaling:=FALSE;
END_METHOD

END_FUNCTION_BLOCK

// LowLevel_Algoritms/algoritms/MvProtection
	{attribute 'symbol' := 'none'}
FUNCTION_BLOCK MvProtection EXTENDS BaseProtection
VAR_INPUT
	sw:REFERENCE TO SectionSwitch;
	delay:TimeParametr(table:=ADR(objectTable));
END_VAR
VAR_OUTPUT
END_VAR
VAR
	timer:ton;
END_VAR

SUPER^();
timer(in:= ((sw.onStatus<> statusDualInput.STATUS_ON) AND (ai.TokStatora.value < 240)), pt:=delay.Value);
IF timer.Q THEN
	signaling:=TRUE;
ELSE
	signaling:=FALSE;
END_IF

METHOD PUBLIC reset
VAR_INPUT
END_VAR
SUPER^.reset();
signaling:=FALSE;
END_METHOD

END_FUNCTION_BLOCK

// lowLevel_ecl/im/sectionSwitch/SectionSwitch
	{attribute 'symbol' := 'none'}
FUNCTION_BLOCK SectionSwitch EXTENDS DualStateSwitch
VAR_INPUT
	basketRolledIn:REFERENCE TO ReliableBit;
	basketRolledOut:REFERENCE TO ReliableBit;
	basketTest:REFERENCE TO ReliableBit;
	
	inLocal: REFERENCE TO ReliableBit;	
	inDistance: REFERENCE TO ReliableBit;
	inVysov: REFERENCE TO ReliableBit;
END_VAR
VAR_OUTPUT
	basketStatus:basketStats;
	local: BOOL;	
	distance: BOOL;
	vysov: BOOL;
END_VAR
VAR
	_noLinks:AloneLogMessage;
	_plakats:UINT;
	Rolled_On_ton: TON:=(pt:=T#2S);
	Rolled_Off_ton: TON:=(pt:=T#2S);
	Rolled_On_R_ton: TON:=(pt:=T#2S);
	Rolled_Off_R_ton: TON:=(pt:=T#2S);

	_basketRolledIn: ReliableBit;
	_basketRolledOut: ReliableBit;
	_basketTest: ReliableBit;
	_basketRolledIn_izm:ReliableBit;
	_basketRolledOut_izm: ReliableBit;
END_VAR
VAR CONSTANT
	cmd_setPlakat:UINT:=4;
	cmd_resetPlakat:UINT:=5;
END_VAR

SUPER^();

IF NOT __ISVALIDREF(basketRolledIn) AND NOT __ISVALIDREF(basketRolledOut) THEN
	basketStatus:=basketStats.BASKET_NOTDEFINED;
	_noLinks.write(CmpLog.LogClass.LOG_ERROR,name,'wrong basket links: ');
ELSE
	IF __ISVALIDREF(basketRolledIn) THEN
		_basketRolledIn:=basketRolledIn;
	ELSE
		_basketRolledIn:=basketRolledOut;
		_basketRolledIn.setValue(NOT _basketRolledIn.value);
	END_IF
	
	IF __ISVALIDREF(basketRolledOut) THEN
		_basketRolledOut:=basketRolledOut;
	ELSE
		_basketRolledOut:=basketRolledIn;
		_basketRolledOut.setValue(NOT _basketRolledOut.value);	
	END_IF
	
	IF __ISVALIDREF(basketTest) THEN
		_basketTest:=basketTest;
	ELSE
		_basketTest.setReliability(TRUE);
		_basketTest.setValue(FALSE);
	END_IF
	
	Rolled_On_ton (IN:=(_basketRolledIn_izm.value <> _basketRolledIn.value));
	Rolled_On_R_ton (IN:=(_basketRolledIn_izm.reliability <> _basketRolledIn.reliability));
	
	Rolled_Off_ton (IN:=(_basketRolledOut_izm.value <> _basketRolledOut.value));
	Rolled_Off_R_ton (IN:=(_basketRolledOut_izm.reliability <> _basketRolledOut.reliability));
	
	IF	Rolled_On_ton.Q THEN
		_basketRolledIn_izm.setValue (_basketRolledIn.value);
	END_IF
	
	IF	Rolled_On_R_ton.Q THEN
		_basketRolledIn_izm.setReliability (_basketRolledIn.reliability);
	END_IF
	
	IF	Rolled_Off_ton.Q THEN
		_basketRolledOut_izm.setValue (_basketRolledOut.value);
	END_IF
	
	IF	Rolled_Off_R_ton.Q THEN
		_basketRolledOut_izm.setReliability (_basketRolledOut.reliability);
	END_IF
	
	IF _basketRolledIn_izm.reliability AND _basketRolledOut_izm.reliability AND _basketTest.reliability THEN
		IF (BOOL_TO_INT(_basketRolledIn_izm.value)+BOOL_TO_INT(_basketRolledOut_izm.value)+BOOL_TO_INT(_basketTest.value))=1 THEN
			IF _basketRolledIn_izm.value THEN
				basketStatus:=basketStats.BASKET_ROLLEDIN;
			ELSIF _basketRolledOut_izm.value THEN
				basketStatus:=basketStats.BASKET_ROLLEDOUT;
			ELSIF _basketTest.value THEN
				basketStatus:=basketStats.BASKET_TEST;
			END_IF
		ELSE			
			basketStatus:=basketStats.BASKET_ERROR;
		END_IF
	ELSE
		basketStatus:=basketStats.BASKET_NOTDEFINED;
	END_IF
END_IF

local:=checkArg(inLocal);	
distance:=checkArg(inDistance);
vysov := checkArg(inVysov);

METHOD on
VAR_INPUT
END_VAR
IF (_plakats=0) THEN
	SUPER^.on();
ELSE
	setCmd(nCmd:=cmd_on);
	errorCommand();
END_IF
END_METHOD

METHOD PROTECTED processCmd;
VAR_INPUT
	cmd:UINT;
	sender:UINT;
	parametr:UINT;
END_VAR
SUPER^.processCmd(cmd,sender,parametr);
CASE cmd OF
	cmd_setPlakat :setPlakat(parametr);
	cmd_resetPlakat :resetPlakat(parametr);
END_CASE
END_METHOD

METHOD PUBLIC resetPlakat
VAR_INPUT
	plakat:UINT;
END_VAR
setCmd(cmd_ResetPlakat);
_plakats:=_plakats AND (NOT plakat);
resetCommand();
END_METHOD

METHOD PUBLIC setPlakat
VAR_INPUT
	Plakat:UINT ;
END_VAR
setCmd(cmd_setPlakat);
_plakats:=_plakats OR Plakat;
resetCommand();
END_METHOD

METHOD PUBLIC writeImStatus
VAR_INPUT
END_VAR
SUPER^.writeImStatus();
statusSet.setBits(8,10,basketStatus);
statusSet.setBits(11,14,_plakats);
statusSet.setBit(5,local);
statusSet.setBit(6,distance);
statusSet.setBit(7,vysov);
END_METHOD

END_FUNCTION_BLOCK

// lowLevel_ecl/im/BaseIms/DualStateSwitch
	{attribute 'symbol' := 'none'}
FUNCTION_BLOCK DualStateSwitch EXTENDS DualStateIm
VAR_INPUT
	
	commandTime:TIME:=T#5S;
	waitStatus:TIME:=T#5S;
END_VAR
VAR_OUTPUT

END_VAR
VAR
	_StatusErrorTimer:TON;
	_resetOutputs:TON;
END_VAR
VAR CONSTANT
	cmd_on:WORD:=1;
	cmd_off:WORD:=2;
END_VAR

SUPER^();

METHOD on
VAR_INPUT
END_VAR
setCmd(nCmd:=cmd_on);
_StatusErrorTimer(IN:=FALSE);
_StatusErrorTimer.IN:=TRUE;
_resetOutputs(In:=FALSE);
_resetOutputs.IN:=TRUE;
SUPER^.on();
END_METHOD

METHOD PRIVATE resetOutputs:bool
VAR_INPUT
END_VAR
_resetOutputs(PT:=commandTime);

IF (_resetOutputs.Q) THEN
	resetOutputs:=TRUE;
	SUPER^.resetOuts();
END_IF
END_METHOD

//Метод вызывается каждый такт пересчета пока идет выполенение команды.
METHOD PROTECTED onCommandActive
VAR_INPUT
	command:WORD;
END_VAR
CASE command OF
	cmd_on:
		IF resetOutputs() AND (onStatus=statusDualInput.STATUS_ON) THEN
			resetCommand();
			RETURN;
		END_IF
	cmd_off:
		IF resetOutputs() AND (onStatus=statusDualInput.STATUS_OFF) THEN
			resetCommand();
			RETURN;
		END_IF
ELSE
	SUPER^.onCommandActive(command);
	RETURN;
END_CASE

_StatusErrorTimer(PT:=waitStatus);
IF _StatusErrorTimer.Q THEN
		errorCommand();	
END_IF
END_METHOD

METHOD PROTECTED processCmd;
VAR_INPUT
	cmd:UINT;
	sender:UINT;
	parametr:UINT;
END_VAR
SUPER^.processCmd(cmd,sender,parametr);
CASE cmd OF
	cmd_on:on();
	cmd_off:off();
END_CASE
END_METHOD

METHOD PROTECTED resetCommand
VAR_INPUT
END_VAR
SUPER^.resetCommand();
_StatusErrorTimer(IN:=FALSE);
_resetOutputs(In:=FALSE);
END_METHOD

METHOD off
VAR_INPUT
END_VAR
setCmd(nCmd:=cmd_off);
_StatusErrorTimer(IN:=FALSE);
_StatusErrorTimer.IN:=TRUE;
_resetOutputs(In:=FALSE);
_resetOutputs.IN:=TRUE;
SUPER^.off();
END_METHOD

END_FUNCTION_BLOCK

// K1/std12k5/Logic/PPU_Init
	{attribute 'symbol' := 'none'}
FUNCTION_BLOCK PPU_Init EXTENDS Baseim
VAR_INPUT
	
END_VAR
VAR
		AoTrig:F_TRIG;
	ton1: TON;
	ton2: ton;
	Pr_Pvh_r:R_trig;
	Pr_Pvh_f:F_trig;
	Pr_Pms_on_r:R_trig;
	Pr_Pms_off_r:R_trig;
	Mv_pr_on_r:R_trig;
	Mv_pr_off_r:R_trig;
	Krans_On_R:R_trig;
	Krans_Off_R:R_trig;
	dPmg_On_R:R_trig;
	dPmg_Off_R:R_trig;
END_VAR

SUPER^();
ton2(in:=Im.BEAO_Work.Q, pt:=T#3S);
////////////////*РЕЖИМ ЭО*///////////////////////// 
IF 	ton2.Q THEN //выставляем режим экстренного останова
	algmanager.setMode(nMode:=ModeGpa.MODE_EO);
END_IF
////////////*ЗАПУСК АО ОТ ЗАЩИТ*/////////////////////////////
IF 	((protectManager.anyProtectionSignaling() AND NOT((algmanager.mode=ModeGpa.MODE_AO) OR (algmanager.mode=ModeGpa.MODE_EO) OR (algmanager.mode=modegpa.MODE_STOP) OR (algmanager.mode=modegpa.MODE_TESTIM))) OR 
	(protections.p_DGazaNaVhodeNagnetatelja_GPA_STOP.signaling OR protections.p_DGazaNaVyhodeNagnetatelja_GPA_STOP.signaling  OR PROTECTIONS.p_AO_PRU.signaling OR PROTECTIONS.p_AO_fromSHU.signaling)) AND NOT ((algmanager.mode=ModeGpa.TEST_PROTECTIONS) AND (algoritms.Test_P.AO_start.value = 0))   THEN  //выставляем ао при сработке защиты
	algoritms.ao.CanRun:=TRUE;
	algoritms.ao.run();
END_IF
IF 	im.Avtomat_SHU_on.Q THEN
	im.U_Lamp_SHU.on ();
ELSE
	im.U_Lamp_SHU.off ();
END_IF
///////////////*ВЫДАЧА АО И СРАБОТКА ЛАМПОЧКИ АС ПРИ АО И ЭО*//////////////////////////
IF	(algmanager.mode=ModeGpa.MODE_AO) OR (algmanager.mode=ModeGpa.MODE_EO) THEN
	im.AC_Fonar.on();//фонарь включаем
	im.Avary_EGPA.on(); 
	im.AO_Knopka_ind.on ();
ELSE
	im.AC_Fonar.OFf();//фонарь включаем
	im.Avary_EGPA.off(); 
	im.AO_Knopka_ind.off ();
END_IF
////////////////*ЗАПУСК АЛГОРИТМА ВКЛЮЧЕНИЯ ПНС ПРИ ВКЛЮЧЕННОМ МВ*/////////////////////////
IF 	algmanager.mode=modegpa.MODE_STOP AND im.mv.onStatus=statusDualInput.status_on THEN
	algoritms.PNS_ON_MV_.CanRun:=TRUE;
 	algoritms.PNS_ON_MV_.run ();
ELSIF (algmanager.mode=modegpa.MODE_STOP AND im.mv.onStatus=statusDualInput.status_oFF) OR (algmanager.mode <> modegpa.MODE_STOP) THEN
	algmanager.resetAndDisable(alg:=algoritms.PNS_ON_MV_);
END_IF
////////////////*ЗАПУСК ЗАЩИТЫ ПО АО ОТ ШКС04М*/////////////////////////
IF	NOT((algmanager.mode=ModeGpa.MODE_AO) OR (algmanager.mode=ModeGpa.MODE_EO) OR (algmanager.mode=modegpa.MODE_STOP) 
	OR (algmanager.mode=modegpa.MODE_TESTIM) OR (algmanager.mode=modegpa.MODE_NOTDEFINED) OR (algmanager.mode=modegpa.TEST_PROTECTIONS)) THEN
	protections.p_AOKC_SHKC.run();
ELSIF	NOT (algmanager.mode=modegpa.TEST_PROTECTIONS) THEN
	protections.p_AOKC_SHKC.reset();
END_IF;
/////////////*ВЫХОД ИЗ РЕЖИМОВ ОСТАНОВА В РЕЖИМ ГПА ОСТАНОВЛЕН*////////////////////////////
AoTrig(CLK:=algoritms.ao.isRuning OR algoritms.no.isRuning OR ton2.Q); //возврат в режим ГПА остановлен из режимов АО, НО, ЭО
IF 	AoTrig.Q THEN
	algmanager.setMode(nMode:=ModeGpa.MODE_STOP);
END_IF
/////////////*ЗАПУСК НО ОТ КНОПКИ НА ШУ*////////////////////////////
IF	IM.NO_fromSHU.q AND NOT((algmanager.mode=ModeGpa.MODE_AO) OR (algmanager.mode=ModeGpa.MODE_EO)) THEN
	algoritms.no.CanRun:=TRUE;
	ALGORITMS.no.run ();
END_IF
IF	(algmanager.mode=modeGPA.MODE_NO) THEN
	im.NO_Fonar.on ();
ELSE
	im.NO_Fonar.off ();
END_IF
/////////////*ЗАЖИГАЕМ ЛАМПОЧКИ НЕИСПРАВНОСТЕЙ ИЗ РЕЖИМА РАБОТА*////////////////////////////

IF	(algmanager.mode=modeGPA.MODE_WORK_K	) OR (algmanager.mode=modeGPA.MODE_WORK_M) THEN
	IF	(algoritms.ppu.analogSNS ()) OR (protectManager.anyProtectionSignaling ()) OR (algoritms.ppu.Neisp_DI ()) OR (NOT algoritms.ppu.CK_Di ()) THEN
		im.PC_Fonar.on(); 
		im.Neispr_EGPA.on ();
	ELSE
		im.PC_Fonar.off();
		im.Neispr_EGPA.off ();
	END_IF
	im.Work_EGPA.on ();
ELSE
	im.PC_Fonar.off();
	im.Neispr_EGPA.off ();
	im.Work_EGPA.off ();
END_IF
////////////*АЛГОРИТМЫ РАБОТАЮЩИЕ В РЕЖИМЕ ГПА СТОП*/////////////////////////////////
IF	algoritms.ppu.ppuFirst_for_Pusk_Ch OR algoritms.ppu.ppuFirst_for_Pusk_r  AND (algmanager.mode=ModeGpa.MODE_STOP) THEN	
	algoritms.S_AP.CanRun:=TRUE; //алгоритмы пуска
	algoritms.S_PP.CanRun:=TRUE; 
ELSIF	(NOT (algoritms.ppu.ppuFirst_for_Pusk_Ch OR algoritms.ppu.ppuFirst_for_Pusk_r)) AND (algmanager.mode=ModeGpa.MODE_STOP)  THEN
		algoritms.S_AP.CanRun:=FALSE;
		algoritms.S_PP.CanRun:=FALSE;
END_IF;
////////////////////////////////////////
IF	algoritms.ppu.ppuFirst_for_I AND (algmanager.mode=ModeGpa.MODE_STOP) THEN
	algoritms.S_I.CanRun:=TRUE; //алгоритмы имитация пуска
ELSIF	(NOT algoritms.ppu.ppuFirst_for_I) AND (algmanager.mode=ModeGpa.MODE_STOP)  THEN
		algoritms.S_I.CanRun:=FALSE;
END_IF;
////////////////////////////////////////
IF	algoritms.ppu.ppuFirst_for_K AND (algmanager.mode=ModeGpa.MODE_STOP) THEN
	algoritms.S_K.CanRun:=TRUE; //алгоритмы запуска проверки кранов
ELSIF	(NOT algoritms.ppu.ppuFirst_for_I) AND (algmanager.mode=ModeGpa.MODE_STOP)  THEN
		algoritms.S_K.CanRun:=FALSE;
END_IF;		
////////////////////////////////////////
IF	algoritms.ppu.ppuFirst_for_Pms_dPmg	AND (algmanager.mode=ModeGpa.MODE_STOP) THEN
	algoritms.S_dPmg.CanRun:=TRUE; //запуск алгоритмов проверки давление масло смазки и перепад маслогаз
	algoritms.S_Pms.CanRun:=TRUE; 
ELSIF	(NOT algoritms.ppu.ppuFirst_for_Pms_dPmg) AND (algmanager.mode=ModeGpa.MODE_STOP)  THEN
		algoritms.S_dPmg.CanRun:=FALSE; //запуск алгоритмов проверки давление масло смазки и перепад маслогаз
		algoritms.S_Pms.CanRun:=FALSE; 
END_IF;	
////////////////////////////////////////
IF	algoritms.ppu.ppuFirst_for_V_Ch OR algoritms.ppu.ppuFirst_for_V_R AND (algmanager.mode=ModeGpa.MODE_STOP) THEN
	algoritms.S_V.CanRun:=TRUE; //запуск алгоритмов проверки двигателя
ELSIF	(NOT (algoritms.ppu.ppuFirst_for_V_Ch OR algoritms.ppu.ppuFirst_for_V_R)) AND (algmanager.mode=ModeGpa.MODE_STOP)  THEN
		algoritms.S_V.CanRun:=FALSE;
END_IF;	
IF		(algmanager.mode=ModeGpa.MODE_STOP) THEN
		protections.p_TOpornogoPodshipnikaEDT_1.run();
		protections.p_TOpornoYpornogoPodshipnikaEDT_2.run();
		protections.p_TOpornoYpornogoPodshipnikaKolesaRedEDT_3.run();
		protections.p_TOpornoYpornogoPodshipnikaKolesaRedHT_4.run();
		protections.p_TOpornogoPodshipnikaShesterniReduktoraT_5.run();
		protections.p_TOpornogoPodshipnikaReduktoraHT_6.run();
		protections.p_TOpornoYpornogoPodshipnikaNagnetateljaT_7.run();
																										
		protections.p_TOpornoYpornogoPodshipnikaSvobodnogoKoncaNT_8.run();
		protections.p_TYpornogoPodshipnikaRavKolodokHT_9.run();
		protections.p_TYpornogoPodshipnikaNerabKolodokHT_10.run();
		protections.p_TgazaNaVyhodeH.run();
		
	(*Давления*)
		
		protections.p_OsSdvigNagnetatelja_Plus.run();
		protections.p_OsSdvigNagnetatelja_Minus.run();
		
	
	(*Дискретные сигналы *)
		
		
		protections.p_AO_PRU.run();
		protections.p_AO_fromSHU.run();
		algoritms.ppu.run ();
END_IF
////////////////////////////////////////
Pr_Pvh_r (clk:=protections.p_DGazaNaVhodeNagnetatelja_GPA_STOP.isRuning);
Pr_Pvh_f (clk:=protections.p_DGazaNaVhodeNagnetatelja_GPA_STOP.isRuning);

IF	Pr_Pvh_r.Q THEN
	DisableAiLimits(ai := ai.DGazaNaVhodeNagnetatelja,getLimitFlags(AiLimit:=statusAi.Lw));
	DisableAiLimits(ai := ai.DGazaNaVyhodeNagnetatelja,getLimitFlags(AiLimit:=statusAi.Hw));
END_IF
IF	Pr_Pvh_f.Q THEN
	EnableAiLimits(ai := ai.DGazaNaVhodeNagnetatelja,getLimitFlags(AiLimit:=statusAi.Lw));
	EnableAiLimits(ai := ai.DGazaNaVyhodeNagnetatelja,getLimitFlags(AiLimit:=statusAi.Hw));
END_IF
Pr_Pms_on_r (clk:= (protections.p_DavlenijaMasloSmNizkoe.isRuning AND protections.p_DavlenijaMasloSmVysokoe.isRuning));
Pr_Pms_off_r (clk:= NOT (protections.p_DavlenijaMasloSmNizkoe.isRuning AND protections.p_DavlenijaMasloSmVysokoe.isRuning));

IF	Pr_Pms_on_r.Q THEN
	EnableAiLimits(ai := ai.DavlenijaMaslaPosleGNS,getLimitFlags(AiLimit:=statusAi.Lw));
END_IF
IF	Pr_Pms_off_r.Q THEN
	DisableAiLimits(ai := ai.DavlenijaMaslaPosleGNS,getLimitFlags(AiLimit:=statusAi.Lw));
END_IF

Mv_pr_on_r (clk:= (protections.p_mvOff.isRuning));
Mv_pr_off_r (clk:= NOT (protections.p_mvOff.isRuning));

IF	Mv_pr_on_r.Q THEN
	EnableAiLimits(ai := ai.TokStatora,getLimitFlags(AiLimit:=statusAi.lw));
END_IF
IF	Mv_pr_off_r.Q THEN
	DisableAiLimits(ai := ai.TokStatora,getLimitFlags(AiLimit:=statusAi.Lw));
END_IF

Krans_On_R 	(clk:= (protections.p_kran1.isRuning AND protections.p_kran2.isRuning));
Krans_Off_R (clk:= NOT(protections.p_kran1.isRuning AND protections.p_kran2.isRuning));

IF	Krans_On_R.Q THEN
	EnableAiLimits(ai := ai.PerepadDavlenieNaKonfuzore,getLimitFlags(AiLimit:=statusAi.lw));
END_IF
IF	Krans_Off_R.Q THEN
	DisableAiLimits(ai := ai.PerepadDavlenieNaKonfuzore,getLimitFlags(AiLimit:=statusAi.Lw));
END_IF

dPmg_On_R (clk:= (protections.p_PerepadDavlenieMasloGaz.isRuning));
dPmg_Off_R (clk:= NOT (protections.p_PerepadDavlenieMasloGaz.isRuning));

IF	dPmg_On_R.Q THEN
	EnableAiLimits(ai := ai.DavlenijaMaslaPosleNU	,getLimitFlags(AiLimit:=statusAi.lw));
END_IF
IF	dPmg_Off_R.Q THEN
	DisableAiLimits(ai := ai.DavlenijaMaslaPosleNU ,getLimitFlags(AiLimit:=statusAi.Lw));
END_IF
////////////////////////////////////////
ton1 (in:=(algmanager.mode=ModeGpa.MODE_STOP), pt:=T#15S);
////////////////////////////////////////
IF	ton1.Q THEN
	protections.p_DGazaNaVhodeNagnetatelja_GPA_STOP.run ();
	protections.p_DGazaNaVyhodeNagnetatelja_GPA_STOP.run ();
END_IF

END_FUNCTION_BLOCK

// K2/std12k5/Logic/PPU_Init
	{attribute 'symbol' := 'none'}
FUNCTION_BLOCK PPU_Init EXTENDS Baseim
VAR_INPUT
	
END_VAR
VAR
		AoTrig:F_TRIG;
	ton1: TON;
	ton2: ton;
	Pr_Pvh_r:R_trig;
	Pr_Pvh_f:F_trig;
	Pr_Pms_on_r:R_trig;
	Pr_Pms_off_r:R_trig;
	Mv_pr_on_r:R_trig;
	Mv_pr_off_r:R_trig;
	Krans_On_R:R_trig;
	Krans_Off_R:R_trig;
	dPmg_On_R:R_trig;
	dPmg_Off_R:R_trig;
END_VAR

SUPER^();
ton2(in:=Im.BEAO_Work.Q, pt:=T#3S);
////////////////*РЕЖИМ ЭО*///////////////////////// 
IF 	ton2.Q THEN //выставляем режим экстренного останова
	algmanager.setMode(nMode:=ModeGpa.MODE_EO);
END_IF
////////////*ЗАПУСК АО ОТ ЗАЩИТ*/////////////////////////////
IF 	((protectManager.anyProtectionSignaling() AND NOT((algmanager.mode=ModeGpa.MODE_AO) OR (algmanager.mode=ModeGpa.MODE_EO) OR (algmanager.mode=modegpa.MODE_STOP) OR (algmanager.mode=modegpa.MODE_TESTIM))) OR 
	(protections.p_DGazaNaVhodeNagnetatelja_GPA_STOP.signaling OR protections.p_DGazaNaVyhodeNagnetatelja_GPA_STOP.signaling  OR PROTECTIONS.p_AO_PRU.signaling OR PROTECTIONS.p_AO_fromSHU.signaling)) AND NOT ((algmanager.mode=ModeGpa.TEST_PROTECTIONS) AND (algoritms.Test_P.AO_start.value = 0))  THEN  //выставляем ао при сработке защиты
	algoritms.ao.CanRun:=TRUE;
	algoritms.ao.run();
END_IF
IF 	im.Avtomat_SHU_on.Q THEN
	im.U_Lamp_SHU.on ();
ELSE
	im.U_Lamp_SHU.off ();
END_IF
///////////////*ВЫДАЧА АО И СРАБОТКА ЛАМПОЧКИ АС ПРИ АО И ЭО*//////////////////////////
IF	(algmanager.mode=ModeGpa.MODE_AO) OR (algmanager.mode=ModeGpa.MODE_EO) THEN
	im.AC_Fonar.on();//фонарь включаем
	im.Avary_EGPA.on(); 
	im.AO_Knopka_ind.on ();
ELSE
	im.AC_Fonar.OFf();//фонарь включаем
	im.Avary_EGPA.off(); 
	im.AO_Knopka_ind.off ();
END_IF
////////////////*ЗАПУСК АЛГОРИТМА ВКЛЮЧЕНИЯ ПНС ПРИ ВКЛЮЧЕННОМ МВ*/////////////////////////
IF 	algmanager.mode=modegpa.MODE_STOP AND im.mv.onStatus=statusDualInput.status_on THEN
	algoritms.PNS_ON_MV_.CanRun:=TRUE;
 	algoritms.PNS_ON_MV_.run ();
ELSIF (algmanager.mode=modegpa.MODE_STOP AND im.mv.onStatus=statusDualInput.status_oFF) OR (algmanager.mode <> modegpa.MODE_STOP) THEN
	algmanager.resetAndDisable(alg:=algoritms.PNS_ON_MV_);
END_IF
////////////////*ЗАПУСК ЗАЩИТЫ ПО АО ОТ ШКС04М*/////////////////////////
IF	NOT((algmanager.mode=ModeGpa.MODE_AO) OR (algmanager.mode=ModeGpa.MODE_EO) OR (algmanager.mode=modegpa.MODE_STOP) 
	OR (algmanager.mode=modegpa.MODE_TESTIM) OR (algmanager.mode=modegpa.MODE_NOTDEFINED) OR (algmanager.mode=modegpa.TEST_PROTECTIONS)) THEN
	protections.p_AOKC_SHKC.run();
ELSIF	NOT (algmanager.mode=modegpa.TEST_PROTECTIONS) THEN
	protections.p_AOKC_SHKC.reset();
END_IF;
/////////////*ВЫХОД ИЗ РЕЖИМОВ ОСТАНОВА В РЕЖИМ ГПА ОСТАНОВЛЕН*////////////////////////////
AoTrig(CLK:=algoritms.ao.isRuning OR algoritms.no.isRuning OR ton2.Q); //возврат в режим ГПА остановлен из режимов АО, НО, ЭО
IF 	AoTrig.Q THEN
	algmanager.setMode(nMode:=ModeGpa.MODE_STOP);
END_IF
/////////////*ЗАПУСК НО ОТ КНОПКИ НА ШУ*////////////////////////////
IF	IM.NO_fromSHU.q AND NOT((algmanager.mode=ModeGpa.MODE_AO) OR (algmanager.mode=ModeGpa.MODE_EO)) THEN
	algoritms.no.CanRun:=TRUE;
	ALGORITMS.no.run ();
END_IF
IF	(algmanager.mode=modeGPA.MODE_NO) THEN
	im.NO_Fonar.on ();
ELSE
	im.NO_Fonar.off ();
END_IF
/////////////*ЗАЖИГАЕМ ЛАМПОЧКИ НЕИСПРАВНОСТЕЙ ИЗ РЕЖИМА РАБОТА*////////////////////////////

IF	(algmanager.mode=modeGPA.MODE_WORK_K	) OR (algmanager.mode=modeGPA.MODE_WORK_M) THEN
	IF	(algoritms.ppu.analogSNS ()) OR (protectManager.anyProtectionSignaling ()) OR (algoritms.ppu.Neisp_DI ()) OR (NOT algoritms.ppu.CK_Di ()) THEN
		im.PC_Fonar.on(); 
		im.Neispr_EGPA.on ();
	ELSE
		im.PC_Fonar.off();
		im.Neispr_EGPA.off ();
	END_IF
	im.Work_EGPA.on ();
ELSE
	im.PC_Fonar.off();
	im.Neispr_EGPA.off ();
	im.Work_EGPA.off ();
END_IF
////////////*АЛГОРИТМЫ РАБОТАЮЩИЕ В РЕЖИМЕ ГПА СТОП*/////////////////////////////////
IF	algoritms.ppu.ppuFirst_for_Pusk_Ch OR algoritms.ppu.ppuFirst_for_Pusk_r  AND (algmanager.mode=ModeGpa.MODE_STOP) THEN	
	algoritms.S_AP.CanRun:=TRUE; //алгоритмы пуска
	algoritms.S_PP.CanRun:=TRUE; 
ELSIF	(NOT (algoritms.ppu.ppuFirst_for_Pusk_Ch OR algoritms.ppu.ppuFirst_for_Pusk_r)) AND (algmanager.mode=ModeGpa.MODE_STOP)  THEN
		algoritms.S_AP.CanRun:=FALSE;
		algoritms.S_PP.CanRun:=FALSE;
END_IF;
////////////////////////////////////////
IF	algoritms.ppu.ppuFirst_for_I AND (algmanager.mode=ModeGpa.MODE_STOP) THEN
	algoritms.S_I.CanRun:=TRUE; //алгоритмы имитация пуска
ELSIF	(NOT algoritms.ppu.ppuFirst_for_I) AND (algmanager.mode=ModeGpa.MODE_STOP)  THEN
		algoritms.S_I.CanRun:=FALSE;
END_IF;
////////////////////////////////////////
IF	algoritms.ppu.ppuFirst_for_K AND (algmanager.mode=ModeGpa.MODE_STOP) THEN
	algoritms.S_K.CanRun:=TRUE; //алгоритмы запуска проверки кранов
ELSIF	(NOT algoritms.ppu.ppuFirst_for_I) AND (algmanager.mode=ModeGpa.MODE_STOP)  THEN
		algoritms.S_K.CanRun:=FALSE;
END_IF;		
////////////////////////////////////////
IF	algoritms.ppu.ppuFirst_for_Pms_dPmg	AND (algmanager.mode=ModeGpa.MODE_STOP) THEN
	algoritms.S_dPmg.CanRun:=TRUE; //запуск алгоритмов проверки давление масло смазки и перепад маслогаз
	algoritms.S_Pms.CanRun:=TRUE; 
ELSIF	(NOT algoritms.ppu.ppuFirst_for_Pms_dPmg) AND (algmanager.mode=ModeGpa.MODE_STOP)  THEN
		algoritms.S_dPmg.CanRun:=FALSE; //запуск алгоритмов проверки давление масло смазки и перепад маслогаз
		algoritms.S_Pms.CanRun:=FALSE; 
END_IF;	
////////////////////////////////////////
IF	algoritms.ppu.ppuFirst_for_V_Ch OR algoritms.ppu.ppuFirst_for_V_R AND (algmanager.mode=ModeGpa.MODE_STOP) THEN
	algoritms.S_V.CanRun:=TRUE; //запуск алгоритмов проверки двигателя
ELSIF	(NOT (algoritms.ppu.ppuFirst_for_V_Ch OR algoritms.ppu.ppuFirst_for_V_R)) AND (algmanager.mode=ModeGpa.MODE_STOP)  THEN
		algoritms.S_V.CanRun:=FALSE;
END_IF;	
IF		(algmanager.mode=ModeGpa.MODE_STOP) THEN
		protections.p_TOpornogoPodshipnikaEDT_1.run();
		protections.p_TOpornoYpornogoPodshipnikaEDT_2.run();
		protections.p_TOpornoYpornogoPodshipnikaKolesaRedEDT_3.run();
		protections.p_TOpornoYpornogoPodshipnikaKolesaRedHT_4.run();
		protections.p_TOpornogoPodshipnikaShesterniReduktoraT_5.run();
		protections.p_TOpornogoPodshipnikaReduktoraHT_6.run();
		protections.p_TOpornoYpornogoPodshipnikaNagnetateljaT_7.run();
																										
		protections.p_TOpornoYpornogoPodshipnikaSvobodnogoKoncaNT_8.run();
		protections.p_TYpornogoPodshipnikaRavKolodokHT_9.run();
		protections.p_TYpornogoPodshipnikaNerabKolodokHT_10.run();
		protections.p_TgazaNaVyhodeH.run();
		
	(*Давления*)
		
		protections.p_OsSdvigNagnetatelja_Plus.run();
		protections.p_OsSdvigNagnetatelja_Minus.run();
		
	
	(*Дискретные сигналы *)
		
		
		protections.p_AO_PRU.run();
		protections.p_AO_fromSHU.run();
		algoritms.ppu.run ();
END_IF
////////////////////////////////////////
Pr_Pvh_r (clk:=protections.p_DGazaNaVhodeNagnetatelja_GPA_STOP.isRuning);
Pr_Pvh_f (clk:=protections.p_DGazaNaVhodeNagnetatelja_GPA_STOP.isRuning);

IF	Pr_Pvh_r.Q THEN
	DisableAiLimits(ai := ai.DGazaNaVhodeNagnetatelja,getLimitFlags(AiLimit:=statusAi.Lw));
	DisableAiLimits(ai := ai.DGazaNaVyhodeNagnetatelja,getLimitFlags(AiLimit:=statusAi.Hw));
END_IF
IF	Pr_Pvh_f.Q THEN
	EnableAiLimits(ai := ai.DGazaNaVhodeNagnetatelja,getLimitFlags(AiLimit:=statusAi.Lw));
	EnableAiLimits(ai := ai.DGazaNaVyhodeNagnetatelja,getLimitFlags(AiLimit:=statusAi.Hw));
END_IF
Pr_Pms_on_r (clk:= (protections.p_DavlenijaMasloSmNizkoe.isRuning AND protections.p_DavlenijaMasloSmVysokoe.isRuning));
Pr_Pms_off_r (clk:= NOT (protections.p_DavlenijaMasloSmNizkoe.isRuning AND protections.p_DavlenijaMasloSmVysokoe.isRuning));

IF	Pr_Pms_on_r.Q THEN
	EnableAiLimits(ai := ai.DavlenijaMaslaPosleGNS,getLimitFlags(AiLimit:=statusAi.Lw));
END_IF
IF	Pr_Pms_off_r.Q THEN
	DisableAiLimits(ai := ai.DavlenijaMaslaPosleGNS,getLimitFlags(AiLimit:=statusAi.Lw));
END_IF

Mv_pr_on_r (clk:= (protections.p_mvOff.isRuning));
Mv_pr_off_r (clk:= NOT (protections.p_mvOff.isRuning));

IF	Mv_pr_on_r.Q THEN
	EnableAiLimits(ai := ai.TokStatora,getLimitFlags(AiLimit:=statusAi.lw));
END_IF
IF	Mv_pr_off_r.Q THEN
	DisableAiLimits(ai := ai.TokStatora,getLimitFlags(AiLimit:=statusAi.Lw));
END_IF

Krans_On_R 	(clk:= (protections.p_kran1.isRuning AND protections.p_kran2.isRuning));
Krans_Off_R (clk:= NOT(protections.p_kran1.isRuning AND protections.p_kran2.isRuning));

IF	Krans_On_R.Q THEN
	EnableAiLimits(ai := ai.PerepadDavlenieNaKonfuzore,getLimitFlags(AiLimit:=statusAi.lw));
END_IF
IF	Krans_Off_R.Q THEN
	DisableAiLimits(ai := ai.PerepadDavlenieNaKonfuzore,getLimitFlags(AiLimit:=statusAi.Lw));
END_IF

dPmg_On_R (clk:= (protections.p_PerepadDavlenieMasloGaz.isRuning));
dPmg_Off_R (clk:= NOT (protections.p_PerepadDavlenieMasloGaz.isRuning));

IF	dPmg_On_R.Q THEN
	EnableAiLimits(ai := ai.DavlenijaMaslaPosleNU	,getLimitFlags(AiLimit:=statusAi.lw));
END_IF
IF	dPmg_Off_R.Q THEN
	DisableAiLimits(ai := ai.DavlenijaMaslaPosleNU ,getLimitFlags(AiLimit:=statusAi.Lw));
END_IF
////////////////////////////////////////
ton1 (in:=(algmanager.mode=ModeGpa.MODE_STOP), pt:=T#15S);
////////////////////////////////////////
IF	ton1.Q THEN
	protections.p_DGazaNaVhodeNagnetatelja_GPA_STOP.run ();
	protections.p_DGazaNaVyhodeNagnetatelja_GPA_STOP.run ();
END_IF

END_FUNCTION_BLOCK

// K1/std12k5/Logic/Synch_Rejims
	{attribute 'symbol' := 'none'}
FUNCTION_BLOCK Synch_Rejims EXTENDS BaseAlgoritm
VAR_INPUT
END_VAR
VAR_OUTPUT
	
	
END_VAR
VAR
	
	ton1:ton ;
	ton2:ton ;
	ton3:ton ;
END_VAR

SUPER^();

IF	((algmanager.mode=ModeGpa.MODE_STOP) OR (algmanager.mode=ModeGpa.MODE_WORK_K) OR (algmanager.mode=ModeGpa.MODE_WORK_M)) AND MasterOPC_ST THEN
	IF	NOT im.Synch_rej_K1_Meandr.Q THEN
		im.Synch_rej_K1_Meandr.on ();
	END_IF
	IF 	im.Synch_rej_K1_Meandr.Q THEN
		im.Synch_rej_K1_Meandr.off();
	END_IF
	ton1(IN:=FALSE);
	ton2(IN:=FALSE);
	ton3(IN:=FALSE);
ELSE
	im.Synch_rej_K1_Meandr.off();
	IF	((NOT ((algmanager.mode=ModeGpa.MODE_STOP) AND ((im.kran1.onStatus=statusDualInput.status_off) AND (im.kran2.onStatus=statusDualInput.status_off)  AND 
			(im.mv.onStatus=statusDualInput.status_off)))) AND (NOT (((algmanager.mode=ModeGpa.MODE_WORK_K) OR (algmanager.mode=ModeGpa.MODE_WORK_M)) AND ((im.kran1.onStatus=statusDualInput.status_on) AND (im.kran2.onStatus=statusDualInput.status_on)  AND 
			(im.mv.onStatus=statusDualInput.status_on))))) AND NOT MasterOPC_ST THEN
		ton1(IN:=im.Synch_rej_K1.Q, pt:=T#5S); 
		ton2(IN:=(NOT im.Synch_rej_K1.Q), pt:=T#5S);
		ton3(In:= (NOT (ton1.Q OR ton2.Q)), pt:=T#10S);
	ELSIF	(((algmanager.mode=ModeGpa.MODE_STOP) AND NOT((im.kran1.onStatus=statusDualInput.status_on) AND (im.kran2.onStatus=statusDualInput.status_on)  AND 
			(im.mv.onStatus=statusDualInput.status_on))) OR (((algmanager.mode=ModeGpa.MODE_WORK_K) OR (algmanager.mode=ModeGpa.MODE_WORK_M)) AND 
			((im.kran1.onStatus=statusDualInput.status_on) AND (im.kran2.onStatus=statusDualInput.status_on)  AND 
			(im.mv.onStatus=statusDualInput.status_on)))) AND NOT MasterOPC_ST THEN
			ton1(IN:=FALSE);
			ton2(IN:=FALSE);
			ton3(IN:=FALSE);
	END_IF
END_IF

IF	(ton3.Q AND (im.kran1.onStatus=statusDualInput.status_on) AND (im.kran2.onStatus=statusDualInput.status_on)  AND (im.mv.onStatus=statusDualInput.status_on)) THEN
	IF 	im.kran6.onStatus=statusDualInput.status_on THEN
		algManager.setMode(nMode:=ModeGpa.MODE_WORK_K);
	ELSIF	im.kran6.onStatus=statusDualInput.status_off THEN
		algManager.setMode(nMode:=ModeGpa.MODE_WORK_M);
		algoritms.S_Vibr.CanRun:=TRUE;
		algoritms.S_Vibr.run ();
	END_IF
	protections.p_DavlenijaMasloSmNizkoe.run();
	protections.p_DavlenijaMasloSmVysokoe.run ();
	protections.p_mvOff.run (); //включаем защиты по МВ и возбудителю
	protections.p_OFFAvarSwitch.run();
	protections.p_RegVozbOff.run();
	protections.p_PerepadDavlenieMasloGaz.run();
	protections.p_PerepadDavlenieMasloGaz_Less100.run ();
	protections.p_DGazaNaVhodeNagnetatelja_GPA_STOP.reset ();
	protections.p_DGazaNaVyhodeNagnetatelja_GPA_STOP.reset ();
	algoritms.autoNu_2.CanRun:=TRUE;
	algoritms.autoNu_2.run ();
	algoritms.autoPns.CanRun :=TRUE;
	algoritms.autoPns.run();
	algoritms.S_AutoAVOM.CanRun:=TRUE;
	//protections.p_DGazaNaVhodeNagnetatelja.run ();
	protections.p_DGazaNaVyhodeNagnetatelja.run ();
	algoritms.Kr6_Move.canrun:=TRUE;
	algoritms.Kr6_Move.run();
	protections.p_kran1.run();
	protections.p_kran2.run();
ELSIF	(ton3.Q AND (im.kran1.onStatus=statusDualInput.status_off) AND (im.kran2.onStatus=statusDualInput.status_off)AND (im.mv.onStatus=statusDualInput.status_off)) THEN
		protections.p_mvOff.reset ();
		protections.p_OFFAvarSwitch.reset();
		protections.p_RegVozbOff.reset ();
		protections.p_kran1.reset ();
		protections.p_kran2.reset ();
		protections.p_PerepadDavlenieMasloGaz.reset();
		protections.p_PerepadDavlenieMasloGaz_Less100.reset();
		protections.p_DGazaNaVhodeNagnetatelja_GPA_STOP.run ();
		protections.p_DGazaNaVyhodeNagnetatelja_GPA_STOP.run ();
		//protections.p_DGazaNaVhodeNagnetatelja.reset ();
		protections.p_DGazaNaVyhodeNagnetatelja.reset ();
		protections.p_DavlenijaMasloSmNizkoe.reset ();
		protections.p_DavlenijaMasloSmVysokoe.reset ();
		algManager.setMode(nMode:=ModeGpa.MODE_STOP);
END_IF

END_FUNCTION_BLOCK

// K2/std12k5/Logic/Synch_Rejims
	{attribute 'symbol' := 'none'}
FUNCTION_BLOCK Synch_Rejims EXTENDS BaseAlgoritm
VAR_INPUT
END_VAR
VAR_OUTPUT
	
	
END_VAR
VAR
	
	ton1:ton ;
	ton2:ton ;
	ton3:ton ;
END_VAR

SUPER^();

IF	((algmanager.mode=ModeGpa.MODE_STOP) OR (algmanager.mode=ModeGpa.MODE_WORK_K) OR (algmanager.mode=ModeGpa.MODE_WORK_M)) AND MasterOPC_ST THEN
	IF	NOT im.Synch_rej_K1_Meandr.Q THEN
		im.Synch_rej_K1_Meandr.on ();
	END_IF
	IF 	im.Synch_rej_K1_Meandr.Q THEN
		im.Synch_rej_K1_Meandr.off();
	END_IF
	ton1(IN:=FALSE);
	ton2(IN:=FALSE);
	ton3(IN:=FALSE);
ELSE
	im.Synch_rej_K1_Meandr.off();
	IF	((NOT ((algmanager.mode=ModeGpa.MODE_STOP) AND ((im.kran1.onStatus=statusDualInput.status_off) AND (im.kran2.onStatus=statusDualInput.status_off)  AND 
			(im.mv.onStatus=statusDualInput.status_off)))) AND (NOT (((algmanager.mode=ModeGpa.MODE_WORK_K) OR (algmanager.mode=ModeGpa.MODE_WORK_M)) AND ((im.kran1.onStatus=statusDualInput.status_on) AND (im.kran2.onStatus=statusDualInput.status_on)  AND 
			(im.mv.onStatus=statusDualInput.status_on))))) AND NOT MasterOPC_ST THEN
		ton1(IN:=im.Synch_rej_K1.Q, pt:=T#5S); 
		ton2(IN:=(NOT im.Synch_rej_K1.Q), pt:=T#5S);
		ton3(In:= (NOT (ton1.Q OR ton2.Q)), pt:=T#10S);
	ELSIF	(((algmanager.mode=ModeGpa.MODE_STOP) AND NOT((im.kran1.onStatus=statusDualInput.status_on) AND (im.kran2.onStatus=statusDualInput.status_on)  AND 
			(im.mv.onStatus=statusDualInput.status_on))) OR (((algmanager.mode=ModeGpa.MODE_WORK_K) OR (algmanager.mode=ModeGpa.MODE_WORK_M)) AND 
			((im.kran1.onStatus=statusDualInput.status_on) AND (im.kran2.onStatus=statusDualInput.status_on)  AND 
			(im.mv.onStatus=statusDualInput.status_on)))) AND NOT MasterOPC_ST THEN
			ton1(IN:=FALSE);
			ton2(IN:=FALSE);
			ton3(IN:=FALSE);
	END_IF
END_IF

IF	(ton3.Q AND (im.kran1.onStatus=statusDualInput.status_on) AND (im.kran2.onStatus=statusDualInput.status_on)  AND (im.mv.onStatus=statusDualInput.status_on)) THEN
	IF 	im.kran6.onStatus=statusDualInput.status_on THEN
		algManager.setMode(nMode:=ModeGpa.MODE_WORK_K);
	ELSIF	im.kran6.onStatus=statusDualInput.status_off THEN
		algManager.setMode(nMode:=ModeGpa.MODE_WORK_M);
		algoritms.S_Vibr.CanRun:=TRUE;
		algoritms.S_Vibr.run ();
	END_IF
	protections.p_DavlenijaMasloSmNizkoe.run();
	protections.p_DavlenijaMasloSmVysokoe.run ();
	protections.p_mvOff.run (); //включаем защиты по МВ и возбудителю
	protections.p_OFFAvarSwitch.run();
	protections.p_RegVozbOff.run();
	protections.p_PerepadDavlenieMasloGaz.run();
	protections.p_PerepadDavlenieMasloGaz_Less100.run ();
	protections.p_DGazaNaVhodeNagnetatelja_GPA_STOP.reset ();
	protections.p_DGazaNaVyhodeNagnetatelja_GPA_STOP.reset ();
	algoritms.autoNu_2.CanRun:=TRUE;
	algoritms.autoNu_2.run ();
	algoritms.autoPns.CanRun :=TRUE;
	algoritms.autoPns.run();
	algoritms.S_AutoAVOM.CanRun:=TRUE;
	//protections.p_DGazaNaVhodeNagnetatelja.run ();
	protections.p_DGazaNaVyhodeNagnetatelja.run ();
	algoritms.Kr6_Move.canrun:=TRUE;
	algoritms.Kr6_Move.run();
	protections.p_kran1.run();
	protections.p_kran2.run();
ELSIF	(ton3.Q AND (im.kran1.onStatus=statusDualInput.status_off) AND (im.kran2.onStatus=statusDualInput.status_off)AND (im.mv.onStatus=statusDualInput.status_off)) THEN
		protections.p_mvOff.reset ();
		protections.p_OFFAvarSwitch.reset();
		protections.p_RegVozbOff.reset ();
		protections.p_kran1.reset ();
		protections.p_kran2.reset ();
		protections.p_PerepadDavlenieMasloGaz.reset();
		protections.p_PerepadDavlenieMasloGaz_Less100.reset();
		protections.p_DGazaNaVhodeNagnetatelja_GPA_STOP.run ();
		protections.p_DGazaNaVyhodeNagnetatelja_GPA_STOP.run ();
		//protections.p_DGazaNaVhodeNagnetatelja.reset ();
		protections.p_DGazaNaVyhodeNagnetatelja.reset ();
		protections.p_DavlenijaMasloSmNizkoe.reset ();
		protections.p_DavlenijaMasloSmVysokoe.reset ();
		algManager.setMode(nMode:=ModeGpa.MODE_STOP);
END_IF

END_FUNCTION_BLOCK

// K1/std12k5/ProtectionManager
	{attribute 'symbol' := 'none'}
FUNCTION_BLOCK ProtectionManager EXTENDS BaseAlgoritmsManager
VAR_INPUT
END_VAR
VAR_OUTPUT
	
END_VAR
VAR

END_VAR

SUPER^();

METHOD PUBLIC anyProtectionSignaling : BOOL
VAR_INPUT
END_VAR
VAR
		curObject:POINTER TO BaseObject;
		IcurProtection:IProtection;
END_VAR

curObject:=	objectTable.head;
IF curObject<>0 THEN
	REPEAT
		IF (__QUERYINTERFACE(curObject^,IcurProtection)) THEN
			IF IcurProtection.Signaling THEN
				anyProtectionSignaling:=TRUE;
				RETURN;
			END_IF	
		END_IF;
		curObject:=curObject^.getNext();
	UNTIL curObject=0
	END_REPEAT;
END_IF;
anyProtectionSignaling:=FALSE;
END_METHOD

END_FUNCTION_BLOCK

// K2/std12k5/ProtectionManager
	{attribute 'symbol' := 'none'}
FUNCTION_BLOCK ProtectionManager EXTENDS BaseAlgoritmsManager
VAR_INPUT
END_VAR
VAR_OUTPUT
	
END_VAR
VAR

END_VAR

SUPER^();

METHOD PUBLIC anyProtectionSignaling : BOOL
VAR_INPUT
END_VAR
VAR
		curObject:POINTER TO BaseObject;
		IcurProtection:IProtection;
END_VAR

curObject:=	objectTable.head;
IF curObject<>0 THEN
	REPEAT
		IF (__QUERYINTERFACE(curObject^,IcurProtection)) THEN
			IF IcurProtection.Signaling THEN
				anyProtectionSignaling:=TRUE;
				RETURN;
			END_IF	
		END_IF;
		curObject:=curObject^.getNext();
	UNTIL curObject=0
	END_REPEAT;
END_IF;
anyProtectionSignaling:=FALSE;
END_METHOD

END_FUNCTION_BLOCK

// lowLevel_ecl/Common/fb/RsRTrig
FUNCTION_BLOCK RsRTrig
VAR_INPUT
	set:BOOL;
	reset:BOOL;
END_VAR
VAR_OUTPUT
	Q:BOOL;
	Qset:BOOL;
END_VAR
VAR
	rsTrig:RS;
	rTrig:R_TRIG;
END_VAR

rsTrig(SET:=set,RESET1:=reset,Q1=>rTrig.CLK);
rTrig(Q=>Q);
Qset:=set;

END_FUNCTION_BLOCK

// lowLevel_ecl/Common/fb/unpackTime
FUNCTION_BLOCK unpackTime
VAR_INPUT
	in: TIME;
END_VAR
VAR_OUTPUT
	hours:UINT;
	mins:UINT;
	sec:UINT;
	msec:UINT;
END_VAR
VAR
END_VAR
VAR_TEMP
	curTime:DWORD;
END_VAR

curTime:=TIME_TO_DWORD(in);
msec:=UDINT_TO_UINT(curTime MOD 1000);
curTime:=curTime / 1000;

sec:=UDINT_TO_UINT(curTime MOD 60);
curTime:=curTime / 60;

mins:=UDINT_TO_UINT(curTime MOD 60);
curTime:=curTime/60;

hours:=UDINT_TO_UINT(curTime);

END_FUNCTION_BLOCK

// lowLevel_ecl/Common/parameters/AnalogParameter/AnalogParametr
	{attribute 'symbol' := 'none'}
FUNCTION_BLOCK AnalogParametr EXTENDS BaseAnalogParametr
VAR_INPUT
END_VAR
VAR_OUTPUT
END_VAR
VAR
END_VAR

SUPER^();

METHOD PROTECTED processCmd;
VAR_INPUT
	cmd:UINT;
	sender:UINT;
	parametr:UINT;
END_VAR
CASE cmd OF
	cmd_ChangeValue:setValue(newValue);
END_CASE
END_METHOD

METHOD PROTECTED readPersistent
VAR_INPUT
END_VAR
value:=FPU.StrToReal(readValue());
END_METHOD

METHOD PUBLIC setValue
VAR_INPUT
	newValue:REAL;
END_VAR
setCmd(cmd_ChangeValue);
IF isValidValue(newValue) THEN
	Value:=newValue;

	SaveToFile();
	resetCommand();
ELSE
	errorCommand();
END_IF
END_METHOD

METHOD PROTECTED writePersistent
VAR_INPUT
END_VAR
writeValue(value:=FPU.RealToStr(value),comment:='value');
END_METHOD

END_FUNCTION_BLOCK

// lowLevel_ecl/Common/parameters/AnalogParameter/BaseAnalogParametr
	{attribute 'symbol' := 'none'}
FUNCTION_BLOCK BaseAnalogParametr EXTENDS BaseIm IMPLEMENTS IAnalogParameter
VAR_INPUT
		{attribute 'symbol' := 'readwrite'}
	newValue:REAL;	
	
	minVal:REAL:=RNaN();
	maxVal:REAL:=RNaN();
	maxStep:REAL:=RNaN();
END_VAR
VAR_OUTPUT
		{attribute 'symbol' := 'read'}
	Value:REAL;
END_VAR
VAR
	
END_VAR
VAR CONSTANT
	cmd_ChangeValue:WORD:=1;
END_VAR

SUPER^();

METHOD getValue : Real
VAR_INPUT
END_VAR
getValue:=Value;
END_METHOD

METHOD PROTECTED isValidValue : BOOL;
VAR_INPUT
	newValue:REAL;
END_VAR
IF NOT FPU.IsRealNaN(minVal) THEN
	IF newValue<minVal THEN
		isValidValue:=FALSE;
		RETURN;
	END_IF
END_IF

IF NOT FPU.IsRealNaN(maxVal) THEN
	IF newValue>maxVal THEN
		isValidValue:=FALSE;
		RETURN;
	END_IF
END_IF

IF NOT fpu.IsRealNaN(maxStep) THEN
	IF rABS(Value-newValue)>maxStep THEN
		isValidValue:=FALSE;
		RETURN;
	END_IF
END_IF

isValidValue:= TRUE;
END_METHOD

METHOD PUBLIC setValue
VAR_INPUT
	newValue:REAL;
END_VAR
END_METHOD

END_FUNCTION_BLOCK

// lowLevel_ecl/Common/parameters/AnalogParameter/IAnalogParameter
INTERFACE IAnalogParameter EXTENDS IAnalogValue

METHOD setValue
VAR_INPUT
	newValue:REAL;
END_VAR
END_METHOD

END_INTERFACE

// lowLevel_ecl/Common/parameters/AnalogParameter/IAnalogValue
INTERFACE IAnalogValue

METHOD getValue : Real
VAR_INPUT
END_VAR
END_METHOD

END_INTERFACE

// lowLevel_ecl/Common/parameters/AnalogParameter/AnalogParametrDinamic
	{attribute 'symbol' := 'none'}
FUNCTION_BLOCK AnalogParametrDinamic EXTENDS BaseAnalogParametr
VAR_INPUT
END_VAR
VAR_OUTPUT
END_VAR
VAR
	
END_VAR

SUPER^();

METHOD PROTECTED processCmd;
VAR_INPUT
	cmd:UINT;
	sender:UINT;
	parametr:UINT;
END_VAR
CASE cmd OF	
	cmd_ChangeValue:
		setCmd(cmd_ChangeValue);
		IF isValidValue(newValue) THEN
			setValue(newValue);
			resetCommand();
		ELSE
			errorCommand();
		END_IF
END_CASE
END_METHOD

METHOD PUBLIC setValue
VAR_INPUT
	newValue:REAL;
END_VAR
Value:=newValue;
END_METHOD

END_FUNCTION_BLOCK

// lowLevel_ecl/Common/parameters/AnalogParameter/RefToRealAnalogParameter
	{attribute 'symbol' := 'none'}
FUNCTION_BLOCK RefToRealAnalogParameter IMPLEMENTS IAnalogValue
VAR_INPUT
	input: REFERENCE TO REAL;
END_VAR
VAR_OUTPUT
END_VAR
VAR
END_VAR

METHOD getValue : Real
VAR_INPUT
END_VAR
IF __ISVALIDREF(input) THEN
	GetValue:=input;
ELSE
	GetValue:=RNaN();
END_IF
END_METHOD

END_FUNCTION_BLOCK

// lowLevel_ecl/Common/parameters/question/Question
	{attribute 'symbol' := 'none'}
FUNCTION_BLOCK Question EXTENDS BaseIm
VAR_INPUT
	AnswerVariants:UINT;
END_VAR
VAR_OUTPUT
	answer:Answers;
END_VAR
VAR
	Asked:UINT;
	resetAns:TON:=(PT:=T#1S);
	_needResetAns:BOOL;
END_VAR
VAR CONSTANT
	cmd_answer:UINT:=1;
END_VAR

SUPER^();
resetAns();
IF _needResetAns AND resetAns.Q THEN
	reset();
END_IF

METHOD PUBLIC ask : Answers
VAR_INPUT
END_VAR
IF Asked=0 THEN
	Asked:=AnswerVariants;
	answer:=Answers.ANS_NONE;	
END_IF
ask:=answer;
END_METHOD

METHOD PROTECTED processCmd;
VAR_INPUT
	cmd:UINT;
	sender:UINT;
	parametr:UINT;
END_VAR
CASE cmd OF
	cmd_answer:reseiveAnswer(rAnswer:=parametr);
END_CASE
END_METHOD

METHOD PROTECTED reseiveAnswer
VAR_INPUT
	rAnswer:Answers;
END_VAR
setCmd(nCmd:=cmd_answer);
IF Asked<>0 THEN
	answer:=rAnswer;
	resetCommand();
	
	resetAns(in:=FALSE);
	resetAns.IN:=TRUE;
	_needResetAns:=FALSE;
	
ELSE
	errorCommand();
END_IF
END_METHOD

METHOD PUBLIC reset
VAR_INPUT
END_VAR
IF resetAns.Q THEN
	Asked:=0;
	answer:=0;
	_needResetAns:=FALSE;
ELSE
	_needResetAns:=TRUE;
END_IF
END_METHOD

METHOD PUBLIC writeImStatus
VAR_INPUT
END_VAR
SUPER^.writeImStatus();
statusSet.setBit(5,answer<>0);
IF answer=0 THEN
	statusSet.setBits(6,14,asked);
ELSE
	statusSet.setBits(6,14,answer);
END_IF
END_METHOD

END_FUNCTION_BLOCK

// lowLevel_ecl/kontroller/baseSources/DOSource
	{attribute 'symbol' := 'none'}
FUNCTION_BLOCK DOSource EXTENDS BaseObject
IMPLEMENTS ISource, IDiscretArchObject
VAR_INPUT
		addr:WORD;
		bits:ARRAY [0..15] OF BOOL;
END_VAR
VAR_OUTPUT
		{attribute 'symbol' := 'read'}
		value:WORD;
END_VAR
VAR
	_imit:BOOL;  
END_VAR
VAR_TEMP
	bitNumber:INT;
END_VAR

value:=0;
FOR bitNumber:=0 TO 15 DO
	value:=value OR (SHL(BOOL_TO_UINT(bits[bitNumber]),bitNumber));
END_FOR

IF NOT imit THEN
	writeData(value:=value);
END_IF

PROPERTY archName : STRING
GET
archName:=name;
END_GET
END_PROPERTY

PROPERTY archReliability : WORD
GET
archReliability:=0;
END_GET
END_PROPERTY

PROPERTY archValue : WORD
GET
archValue:=value;
END_GET
END_PROPERTY

{attribute 'symbol' := 'none'}
PROPERTY imit : BOOL
GET
imit:=_imit;
END_GET
SET
_imit:=imit;
END_SET
END_PROPERTY

METHOD setValue
VAR_INPUT
	val:WORD;
END_VAR
VAR
	i:word;
	unpackedVal:SmartUnpack;
END_VAR
unpackedVal.value:=val;
FOR i:=0 TO 15 DO
bits[i]:=unpackedVal.getBit(start:=i);
END_FOR
END_METHOD

METHOD writeData
VAR_INPUT
	value:WORD;
END_VAR
END_METHOD

END_FUNCTION_BLOCK

// lowLevel_ecl/kontroller/ExecKontrollersComands
FUNCTION ExecKontrollersComands : bool
VAR_INPUT
	CONSTANT table:TableDescriptor;
END_VAR
VAR
	curObject:POINTER TO BaseObject;
	curKontroller:IKontroller;
END_VAR

curObject:=table.head;
IF curObject=0 THEN
	RETURN;
END_IF
REPEAT
	IF (__QUERYINTERFACE(curObject^,curKontroller)) THEN		
		curKontroller.callCommands();
	END_IF;
	curObject:=curObject^.getNext();
	UNTIL curObject=0
END_REPEAT

END_FUNCTION

// lowLevel_ecl/kontroller/extSources/AiMovingSverage
	{attribute 'symbol' := 'none'}
FUNCTION_BLOCK AiMovingSverage EXTENDS AiSource
VAR_INPUT
	ai:REFERENCE TO AISource;
	historyLenght:INT:=30;
	cicleTime:TIME:=T#100MS;
END_VAR
VAR_OUTPUT
END_VAR
VAR
	history:ARRAY [0..maxHistoryLenght-1] OF REAL;
	nextIndex:INT;
	cicleTimer:TON;
END_VAR
VAR CONSTANT
	maxHistoryLenght:INT:=100;
END_VAR

SUPER^();

{attribute 'symbol' := 'none'}
PROPERTY PUBLIC disabledAlarms : BYTE
GET
disabledAlarms:=_disabledAlarms;
END_GET
SET
VAR
END_VAR
VAR
	i:INT;
END_VAR
_disabledAlarms:=disabledAlarms;

ai.disabledAlarms:=_disabledAlarms;
END_SET
END_PROPERTY

METHOD PROTECTED GetData: REAL
VAR_INPUT
END_VAR
VAR_OUTPUT
	o_interval:statusAi;
END_VAR
IF NOT __ISVALIDREF(ai) THEN
	o_interval:=statusAi.NOTDEFINED;
	RETURN;
END_IF

IF NOT fpu.isRealNan(ai.value) THEN
	o_interval:=ai.interval;
ELSE
	o_interval:=statusAi.NOTDEFINED;
	GetData:=value;
	RETURN;
END_IF

cicleTimer(IN:=TRUE,PT:=cicleTime);

IF ai.interval>=statusAi.normal THEN
	IF cicleTimer.Q THEN
		GetData:=value+(ai.value-getLast())/historyLenght;
		writeNext(ai.value);
		cicleTimer(IN:=FALSE);
	ELSE
		GetData:=value;	
	END_IF
ELSE
	GetData:=value;	
END_IF
END_METHOD

METHOD PRIVATE getLast : Real
VAR_INPUT
END_VAR
getLast:=history[nextIndex];
END_METHOD

PROPERTY imit : bool
GET
imit:= FALSE;
END_GET
SET
END_SET
END_PROPERTY

METHOD PRIVATE writeNext
VAR_INPUT
	value:REAL;
END_VAR
history[nextIndex]:=value;
nextIndex:=nextIndex+1;
IF nextIndex>=historyLenght THEN
	nextIndex:=0;
END_IF
END_METHOD

END_FUNCTION_BLOCK

// lowLevel_ecl/kontroller/extSources/TripledAnalog
{attribute 'symbol' := 'none'}
{attribute 'obsolete' := 'Not supported. use MultiAnalog. '} 
FUNCTION_BLOCK TripledAnalog EXTENDS AISource
VAR_INPUT
	input1:REFERENCE TO AISource;
	input2:REFERENCE TO AISource;
	input3:REFERENCE TO AISource;
END_VAR
VAR_OUTPUT
END_VAR
VAR
	maxDelta:REAL:=RNaN();
	inputs:ARRAY[0..2] OF AnalogItem;
END_VAR

SUPER^();

METHOD PROTECTED GetData : Real
VAR_INPUT
END_VAR
VAR_OUTPUT
	o_interval:statusAi;
END_VAR
VAR
	allInvalid:BOOL:=FALSE;
	sumValue:REAL:=0;
	count:INT:=0;
	i:INT;
END_VAR
initArray();
sort();
o_interval:=statusAi.NOTDEFINED;


IF NOT FPU.IsRealNaN(f:=maxDelta) THEN
	IF __ISVALIDREF(inputs[1].input) THEN		
		allInvalid:=TRUE;
		allInvalid:= allInvalid AND NOT validateInputs(midInp:=inputs[1],inp:=inputs[0]);
		allInvalid:= allInvalid AND NOT validateInputs(midInp:=inputs[1],inp:=inputs[2]);
		IF (allInvalid) THEN
			inputs[1].input.notReliable:=TRUE;
		ELSE
			inputs[1].input.notReliable:=FALSE;
		END_IF
	END_IF
END_IF


FOR i:=0 TO 2 DO
	IF __ISVALIDREF(inputs[i].input) THEN
		IF inputs[i].input.interval>=statusAi.normal THEN
			sumValue:=sumValue+inputs[i].input.value;
			count:=count+1;
		END_IF
	END_IF
END_FOR
IF count>0 THEN
	o_interval:=statusAi.normal;
	GetData:=sumValue/count;
END_IF
END_METHOD

PROPERTY imit : bool
GET
imit:= FALSE;
END_GET
SET
END_SET
END_PROPERTY

{attribute 'call_after_init'} 
METHOD PRIVATE initArray
VAR_INPUT
END_VAR
inputs[0].input REF= input1;
inputs[1].input REF= input2;
inputs[2].input REF= input3;
END_METHOD

METHOD PRIVATE compare:bool
VAR_INPUT
	nas1: AnalogItem;
	nas2: AnalogItem;
END_VAR
IF (__ISVALIDREF(nas1.input) AND (NOT __ISVALIDREF (nas2.input))) THEN
	compare:=FALSE;
	RETURN;
END_IF

IF (NOT __ISVALIDREF(nas1.input) AND (__ISVALIDREF (nas2.input))) THEN
	compare:=TRUE;
	RETURN;
END_IF

compare:=FALSE;

IF (__ISVALIDREF(nas1.input) AND __ISVALIDREF (nas2.input)) THEN
	IF (nas1.input.value>nas2.input.value) OR ((nas1.input.interval<statusAi.normal)AND(nas2.input.interval>=statusAi.normal)) THEN
		compare:=TRUE;
	END_IF
END_IF
END_METHOD

METHOD sort
VAR_INPUT
END_VAR
VAR
	i,j:INT;
	item:AnalogItem;
	compareResult:BOOL;
END_VAR
FOR i:=1 TO 2 DO
	item:= inputs[i];  
	j:= i - 1;
	compareResult:=compare(nas1:=inputs[j],nas2:=item);
	WHILE (j >= 0) AND (compareResult) DO    
	   	inputs[j + 1]:= inputs[j];
	 	j:=j-1;
	 	IF j>=0 THEN
			compareResult:=compare(nas1:=inputs[j],nas2:=item);
		END_IF
	END_WHILE;
	inputs[j + 1]:= item;
END_FOR
END_METHOD

METHOD PRIVATE validateInputs: BOOL
VAR_INPUT
	inp:AnalogItem;
	midInp:AnalogItem;
END_VAR
IF __ISVALIDREF(inp.input) THEN
	IF (inp.input.interval>=statusAi.normal)THEN
		IF rABS(inp.input.value-midInp.input.value)>maxDelta THEN
			inp.input.notReliable:=TRUE;
			validateInputs:=FALSE;
		ELSE
			validateInputs:=TRUE;
		END_IF
	ELSE
		validateInputs:=FALSE;
	END_IF 
END_IF
END_METHOD

END_FUNCTION_BLOCK

// lowLevel_ecl/kontroller/extSources/MultiAnalog
{attribute 'symbol' := 'none'}
FUNCTION_BLOCK MultiAnalog EXTENDS AISource
VAR_INPUT
	input1:REFERENCE TO AISource;
	input2:REFERENCE TO AISource;
	input3:REFERENCE TO AISource;
	input4:REFERENCE TO AISource;
	input5:REFERENCE TO AISource;
	input6:REFERENCE TO AISource;
	input7:REFERENCE TO AISource;
	input8:REFERENCE TO AISource;
	input9:REFERENCE TO AISource;
	input10:REFERENCE TO AISource;
	input11:REFERENCE TO AISource;
	input12:REFERENCE TO AISource;
	
	processing:AnalogsProcessing:=	AnalogsProcessing.AVERAGEVALUE;
	
	limits:MultiAnalogLimits:=MultiAnalogLimits.SELF;
	
	maxDelta:REAL:=RNaN();
END_VAR
VAR_OUTPUT
END_VAR
VAR
	
	inputs:ARRAY[0..arrayLength-1] OF AnalogItem;
	arrayMaxIndex:INT;
END_VAR
VAR CONSTANT
	arrayLength:INT:=12;
END_VAR

SUPER^();

METHOD PROTECTED CalkLimits:statusAi
VAR_INPUT

END_VAR
VAR
	validCnt:INT;
	lwCnt:INT;
	hwCnt:INT;
	laCnt:INT;
	haCnt:INT;
END_VAR
CASE limits OF
	MultiAnalogLimits.SELF:
		CalkLimits:=SUPER^.CalkLimits();
		
	MultiAnalogLimits.ALL_INPUTS:
		InputIntervalsCnt(validCnt=>validCnt,lwCnt=>lwCnt,hwCnt=>hwCnt,laCnt=>laCnt,haCnt=>haCnt);
		IF validCnt=0 THEN
			CalkLimits:=statusAi.NOTDEFINED;
			RETURN;
		END_IF
		CalkLimits:=statusAi.normal;
		IF haCnt=validCnt THEN
			CalkLimits:=statusAi.HA;
		ELSIF laCnt=validCnt THEN
			CalkLimits:=statusAi.LA;
		ELSIF (hwCnt>0) OR (haCnt>0) THEN
			CalkLimits:=statusAi.HW;
		ELSIF (lwCnt>0) OR (laCnt>0) THEN
			CalkLimits:=statusAi.LW;
		END_IF
		
	MultiAnalogLimits.ANY_INPUT:
		InputIntervalsCnt(validCnt=>validCnt,lwCnt=>lwCnt,hwCnt=>hwCnt,laCnt=>laCnt,haCnt=>haCnt);	
		IF validCnt=0 THEN
			CalkLimits:=statusAi.NOTDEFINED;
			RETURN;
		END_IF
		CalkLimits:=statusAi.normal;
		IF haCnt>0 THEN
			CalkLimits:=statusAi.HA;
		ELSIF laCnt>0 THEN
			CalkLimits:=statusAi.LA;
		ELSIF hwCnt>0 THEN
			CalkLimits:=statusAi.HW;
		ELSIF lwCnt>0 THEN
			CalkLimits:=statusAi.LW;
		END_IF
END_CASE
END_METHOD

{attribute 'symbol' := 'none'}
PROPERTY PUBLIC disabledAlarms : BYTE
GET
disabledAlarms:=_disabledAlarms;
END_GET
SET
VAR
END_VAR
VAR
	i:INT;
END_VAR
_disabledAlarms:=disabledAlarms;

FOR i:=0 TO arrayMaxIndex DO
	IF __ISVALIDREF(inputs[i].input) THEN
		inputs[i].input.disabledAlarms:=_disabledAlarms;
	END_IF
END_FOR
END_SET
END_PROPERTY

METHOD PROTECTED GetData : Real
VAR_INPUT
END_VAR
VAR_OUTPUT
	o_interval:statusAi;
END_VAR
sort();
o_interval:=statusAi.NOTRELIABLE;

IF NOT checkInputs() THEN
	GetData:=value;
	RETURN;
END_IF

CalcLLHl();

CASE processing OF
	AnalogsProcessing.AVERAGEVALUE:
		IF averageValue(value=>GetData) THEN
			o_interval:=statusAi.normal;
		END_IF
	AnalogsProcessing.MAXVALUE:
		IF maxValue(value=>GetData) THEN
			o_interval:=statusAi.normal;
		END_IF
	AnalogsProcessing.MINVALUE:
		IF minValue(value=>GetData) THEN
			o_interval:=statusAi.normal;
		END_IF		
	AnalogsProcessing.MEDIANVALUE:
		IF medianValue(value=>GetData) THEN
			o_interval:=statusAi.normal;
		END_IF
END_CASE
END_METHOD

PROPERTY imit : bool
GET
imit:= FALSE;
END_GET
SET
END_SET
END_PROPERTY

METHOD PROTECTED onInit
VAR_INPUT
END_VAR
SUPER^.onInit();
initArray();
END_METHOD

METHOD PRIVATE CalcLLHl
VAR_INPUT
END_VAR
VAR_OUTPUT
	
END_VAR
VAR
	i:INT;
END_VAR
LL:=RNaN();
HL:=RNaN();

FOR i:=0 TO arrayMaxIndex DO
	IF __ISVALIDREF(inputs[i].input) THEN
		IF NOT FPU.IsRealNaN(inputs[i].input.LL) THEN
			IF ( inputs[i].input.LL<LL) OR FPU.IsRealNaN(LL) THEN
				LL:=inputs[i].input.LL;
			END_IF
		END_IF
		IF NOT FPU.IsRealNaN(inputs[i].input.HL) THEN
			IF ( inputs[i].input.HL>HL) OR FPU.IsRealNaN(HL) THEN
				Hl:=inputs[i].input.Hl;
			END_IF
		END_IF
	END_IF
END_FOR
END_METHOD

METHOD PRIVATE checkInputs: BOOL
VAR_INPUT
END_VAR
VAR
	controValue:REAL;
	first:INT;
	last:INT;
	valueInvalidated:BOOL;
END_VAR
IF FPU.IsRealNaN(f:=maxDelta) THEN
	checkInputs:=TRUE;
	RETURN;
END_IF

first:=getNextFirstValid(-1);
last:=getNextLastValid(arrayMaxIndex+1);

IF medianValue(value=>controValue) THEN
	REPEAT
		IF (first<0) OR (last<0) THEN //Не осталось достоверных
			checkInputs:=FALSE;
			RETURN;
		END_IF	
		
		valueInvalidated:=rABS(inputs[first].input.value-inputs[last].input.value)>maxDelta;
		
		IF  valueInvalidated THEN
			IF (last-first)<=1 THEN //Осталось только 2 достоверных
				checkInputs:=FALSE;
				RETURN;
			END_IF
			IF rABS(inputs[first].input.value-controValue)>rABS(inputs[last].input.value-controValue) THEN
				inputs[first].input.notReliable:=TRUE;
				first:=getNextFirstValid(first);
			ELSE
				inputs[last].input.notReliable:=TRUE;
				last:=getNextLastValid(last);
			END_IF
		END_IF		
	UNTIL NOT valueInvalidated
	END_REPEAT
END_IF

checkInputs:=TRUE;
END_METHOD

METHOD PROTECTED getNextFirstValid : int //Protected нужен был в Пурпейской
VAR_INPUT
	index:INT;
END_VAR
getNextFirstValid:=index;
REPEAT
	getNextFirstValid:=getNextFirstValid+1;
	IF getNextFirstValid>arrayMaxIndex THEN
		getNextFirstValid:=-1;
		RETURN;
	END_IF				 
UNTIL isValidInput(inputs[getNextFirstValid])
END_REPEAT
END_METHOD

METHOD PROTECTED getNextLastValid : INT //Protected нужен был в Пурпейской
VAR_INPUT
	index:INT;
END_VAR
getNextLastValid:=index;
REPEAT
	getNextLastValid:=getNextLastValid-1;
	IF getNextLastValid<0 THEN
		getNextLastValid:=-1;
		RETURN;
	END_IF
UNTIL isValidInput(inputs[getNextLastValid])
END_REPEAT
END_METHOD

{attribute 'call_after_init'} 
METHOD PRIVATE initArray
VAR_INPUT
END_VAR
inputs[0].input REF= input1;
inputs[1].input REF= input2;
inputs[2].input REF= input3;
inputs[3].input REF= input4;
inputs[4].input REF= input5;
inputs[5].input REF= input6;
inputs[6].input REF= input7;
inputs[7].input REF= input8;
inputs[8].input REF= input9;
inputs[9].input REF= input10;
inputs[10].input REF= input11;
inputs[11].input REF= input12;

arrayMaxIndex:=arrayLength-1;
sort();
WHILE NOT __ISVALIDREF(inputs[arrayMaxIndex].input) DO
	arrayMaxIndex:=arrayMaxIndex-1;
	IF arrayMaxIndex<0 THEN
		RETURN;
	END_IF
END_WHILE
END_METHOD

METHOD PRIVATE InputIntervalsCnt
VAR_INPUT
END_VAR
VAR_OUTPUT
	validCnt:INT;
	lwCnt:INT;
	hwCnt:INT;
	laCnt:INT;
	haCnt:INT;
END_VAR
VAR
	currentIndex:INT;
END_VAR
currentIndex:=getNextFirstValid(-1);
WHILE currentIndex>=0 DO
	validCnt:=validCnt+1;
	CASE inputs[currentIndex].input.interval OF
		statusAi.LW:
			lwCnt:=lwCnt+1;
		statusAi.HW:
			hwCnt:=hwCnt+1;
		statusAi.LA:
			laCnt:=laCnt+1;
		statusAi.HA:
			haCnt:=haCnt+1;
	END_CASE
	currentIndex:=getNextFirstValid(currentIndex);
END_WHILE
END_METHOD

METHOD PRIVATE isValidInput : BOOL
VAR_INPUT
	input:AnalogItem;
END_VAR
isValidInput:=FALSE;
IF  __ISVALIDREF(input.input)THEN
	isValidInput:=input.input.interval>=statusAi.normal;
END_IF
END_METHOD

METHOD PROTECTED readPersistent
VAR_INPUT
END_VAR
SUPER^.readPersistent();
maxDelta:=FPU.StrToReal(readValue());
END_METHOD

METHOD PRIVATE averageValue : BOOL
VAR_INPUT
END_VAR
VAR_OUTPUT
	value:REAL;
END_VAR
VAR
	count:INT:=0;
	i:INT;
	sumValue:REAL:=0;
END_VAR
value:=RNaN();

FOR i:=0 TO arrayMaxIndex DO
	IF isValidInput(inputs[i]) THEN
			sumValue:=sumValue+inputs[i].input.value;
			count:=count+1;
	END_IF
END_FOR

IF count>0 THEN
	averageValue:=TRUE;
	value:=sumValue/count;
END_IF
END_METHOD

METHOD PRIVATE maxValue : BOOL
VAR_INPUT
END_VAR
VAR_OUTPUT
	value:REAL;
END_VAR
VAR
	i:INT;
END_VAR
value:=RNaN();

FOR i:=0 TO arrayMaxIndex DO
	IF isValidInput(inputs[i]) THEN
		IF (FPU.IsRealNaN(value) OR (inputs[i].input.value > value)) THEN
			value:= inputs[i].input.value;
			maxValue:=TRUE;
		END_IF
	END_IF
END_FOR
END_METHOD

METHOD PRIVATE medianValue : BOOL
VAR_INPUT
END_VAR
VAR_OUTPUT
	value:REAL;
END_VAR
VAR
	first:INT;
	last:INT;
END_VAR
first:=-1;
last:=arrayMaxIndex+1;
value:=RNaN();

